// TIA Portal V16 program export: 0 tag tables, 5 data types, 28 data blocks, 30 code blocks (in call order from the OBs), 2 instance data blocks

TYPE "APP"
// stored: IsFailsafeCompliant false
   STRUCT
      PID_ComponenteProporzionale : DInt;
      PID_ComponenteIntegrale : DInt;
      PID_ComponenteDerivativa : DInt;
      Tiro : Int;   // Valore di tiro richiesto: 1-100 => 1-100% Setup 1, 101-200 => 1-100% Setup 2, 0 => Azzera regolatore
      Tiro1 : Int;
      Tiro2 : Int;
      TiroPrecedente : Int;   // Valore di tiro richiesto istante (n-1)
      TiroAppoggio : Int;
      ErroreAttuale : Int;   // Errore istante (n)
      ErrorePrecedente : Int;   // Errore istante (n-1)
      PID_Kp : Int;   // Kp in uso nel PID
      PID_Ki : Int;   // Ki in uso nel PID
      PID_Kd : Int;   // Kd in uso nel PID
      SetpointTiro : Int;   // Valore di setpoint del PID
      SetpointTiroRampa : Int;   // Valore di setpoint del PID iniziale a rampa
      TransitorioInizialeFase1 : Int;   // Indica che si deve eseguire la rampa iniziale (Fase 1)
      TransitorioFase3 : Int;   // Indica che si deve eseguire la rampa da velocita' alta a media (Fase 3)
      TransitorioFase4 : Int;   // Indica che si deve eseguire la rampa da velocita' media a bassa (Fase 4)
      VelocitaRotazione : Int;   // Velocita' di rotazione richiesta
      VelocitaRotazioneFase2 : Int;   // Velocita' di rotazione richiesta durante la Fase 2
      VelocitaRotazioneAppoggio1 : Int;
      VelocitaRotazioneAppoggio2 : Int;
      Fase1OneShoot : Int;   // Indica che sono appena entrato nella fase di traansitorio di accelerazione (Fase 1)
      Fase2OneShoot : Int;   // Indica che sono appena entrato nella fase di transitorio iniziale (Fase 2)
      Fase3OneShoot : Int;   // Indica che sono appena entrato nella fase di transitorio di velocita' alta - media (Fase 3)
      Fase4OneShoot : Int;   // Indica che sono appena entrato nella fase di transitorio di velocita' media - bassa (Fase 4)
      ArrestoRepentinoOneShoot : Int;   // Indica che sono appena entrato nella fase di arresto repentino
      TiroFase1 : Int;   // Indica il tiro nella Fase 1 usato nella Fase 2
      TempIntero : Int;
      Fase : Int;
      BallerinoPrecedente : Array[0..2] of Int;   // Valore del ballerino negli istanti precedenti
      LimiteComponenteIntegrale : Int;   // Limite della componente integrale durante la transizione dalla velocita alta a media (Fase 3) e dalla media a bassa (Fase 4)
      TiroRichiesto : Int;   // Valore di tiro compreso fra 1 e 100 richiesto dalla logica di controllo
      TimerArrestoRepentino : Int;   // Timer per arresto repentino.
      TiroMinimoArrestoRepentino : Int;   // Tiro minimo durante un'arresto repentino
      VariazioneTiro : Int;   // Variazione del tiro film (ballerino)
      TimerFase2 : Int;   // Timer usato nella Fase 2 per arrestare i rulli in caso di rottura film
      TempoRotturaFilm : Int;   // Tempo rottura film in numero di scansioni (1 scansione ogni 30msec)
      TimerFase4 : Int;   // Timer per Fase 4
      TiroMinimoFase4 : Int;   // Tiro minimo durante la Fase 4 di arresto
      PID_Uscita : DInt;   // Valore di uscita del PID
      PrestiroRichiesto : DInt;   // Valore di prestiro richiesto. Valore compreso fra 0 e 500
      PrestiroAppoggio : Real;
   END_STRUCT;
END_TYPE

TYPE "DatiProgramma"
// stored: IsFailsafeCompliant false
   STRUCT
      Wrapping : Bool;   // Wrapping (0=Excluded 1=Included)
      TopLenght : Int;   // Top film lenght
      TopRelease : Int;   // Top carriage release position
      TopDown : Int;   // Top carriage downward to release top film
      Top : Int;   // Top cycle (1=Excluded 2=Before 3=Waterp-2 4=Waterp-3 5=Waterp-4)
      PressurePTime : Int;   // Time for pressure plate downward
      LifterTime : Int;   // Time for pallet lifter upward
      RevOverContrast : Int;   // Revolution over welder contrast
      RopeEndCycle : Byte;   // Rope type at end of cycle (Program)
      Spare4 : Byte;
      RopeTime : Int;   // Delay for rope unit opened
      RevOverClamp : Int;   // Revolution over clamp
      FilmForceFinalRev : Int;   // Film force on the final revolutions
      FilmPrestretchFinalRev : Int;   // Film prestretch on the final revolutions
      ArmSpeed : Int;   // Arm rotation speed (%*10)
      CarriageDown4Top : Int;   // Spool carriage downward for top cycle
      TopDownTime : Int;   // Top carriage downward for top cycle
      LapsUnderTop : Int;   // Revolutions under top film
      Spare6 : Int;   // Spare
      Spare7 : Int;   // Spare
      Spare8 : Int;   // Spare
      Spare9 : Int;   // Spare
      Spare10 : Int;   // Spare
      Spare11 : Int;   // Spare
      Spare12 : Int;   // Spare
      Overlap0_1 : Int := 0;   // Film overlap spool carriage height 0->1
      Height1 : Int := 0;   // Spool carriage height 1 (mm)
      Landmark1 : Bool := false;   // Landmark for spool carriage height 1 (0=Bottom 1=Top)
      Lifter1 : Bool := false;   // Pallet lifter for spool carriage height 1
      SpareBit1H1 : Bool := false;   // Spare bit for spool carriage height 1 (Program)
      Airblower1 : Bool := false;   // Airblower on film tail for spool carriage height 1 (0=Excluded 1=Included)
      NextStep1 : Bool := false;   // Next step for spool carriage height 1 (0=End 1=Next)
      PressureP1 : Bool := false;   // Pressure plate for spool carriage height 1 (0=Excluded 1=Included)
      SpareByte2H1 : Byte := 16#0;   // Spare byte for spool carriage height 1
      Revolution1 : Int := 0;   // Revolutions for spool carriage height 1
      RopeUnit1_1 : Byte := 16#0;   // Rope unit for spool carriage height 1 (1=Excluded 2=Inc 3=Inc during)
      RopeUnit1_2 : Byte := 16#0;   // Rope unit for spool carriage height 1 (1=Excluded 2=Inc 3=Inc during)
      FilmForce1 : Int := 0;   // Film force for spool carriage height 1
      FilmPrestretch1 : Int := 0;   // Film prestretch for spool carriage height 1
      Spare3H1 : Int := 0;   // Spare for spool carriage height 1
      Spare49 : Int := 0;   // Spare
      Spare50 : Int := 0;   // Spare
      Spare51 : Int := 0;   // Spare
      Spare52 : Int := 0;   // Spare
      Spare53 : Int := 0;   // Spare
      Overlap1_2 : Int := 0;   // Film overlap spool carriage height 1->2
      Height2 : Int := 0;   // Spool carriage height 2 (mm)
      Landmark2 : Bool := false;   // Landmark for spool carriage height 2 (0=Bottom 1=Top)
      Lifter2 : Bool := false;   // Pallet lifter for spool carriage height 2
      SpareBit1H2 : Bool := false;   // Spare bit for spool carriage height 2
      Airblower2 : Bool := false;   // Airblower on film tail for spool carriage height 2 (0=Excluded 1=Included)
      NextStep2 : Bool := false;   // Next step for spool carriage height 2 (0=End 1=Next)
      PressureP2 : Bool := false;   // Pressure plate for spool carriage height 2 (0=Excluded 1=Included)
      SpareByte2H2 : Byte := 16#0;   // Spare byte for spool carriage height 2
      Revolution2 : Int := 0;   // Revolutions for spool carriage height 2
      RopeUnit2_1 : Byte := 16#0;   // Rope unit for spool carriage height 2 (1=Excluded 2=Inc 3=Inc during)
      RopeUnit2_2 : Byte := 16#0;   // Rope unit for spool carriage height 2 (1=Excluded 2=Inc 3=Inc during)
      FilmForce2 : Int := 0;   // Film force for spool carriage height 2
      FilmPrestretch2 : Int := 0;   // Film prestretch for spool carriage height 2
      Spare3H2 : Int := 0;   // Spare for spool carriage height 2
      Spare54 : Int := 0;   // Spare
      Spare55 : Int := 0;   // Spare
      Spare56 : Int := 0;   // Spare
      Spare57 : Int := 0;   // Spare
      Spare58 : Int := 0;   // Spare
      Overlap2_3 : Int := 0;   // Film overlap spool carriage height 2->3
      Height3 : Int := 0;   // Spool carriage height 3 (mm)
      Landmark3 : Bool := false;   // Landmark for spool carriage height 3 (0=Bottom 1=Top)
      Lifter3 : Bool := false;   // Pallet lifter for spool carriage height 3
      SpareBit1H3 : Bool := false;   // Spare bit for spool carriage height 3
      Airblower3 : Bool := false;   // Airblower on film tail for spool carriage height 3 (0=Excluded 1=Included)
      NextStep3 : Bool := false;   // Next step for spool carriage height 3 (0=End 1=Next)
      PressureP3 : Bool := false;   // Pressure plate for spool carriage height 3 (0=Excluded 1=Included)
      SpareByte2H3 : Byte := 16#0;   // Spare byte for spool carriage height 3
      Revolution3 : Int := 0;   // Revolutions for spool carriage height 3
      RopeUnit3_1 : Byte := 16#0;   // Rope unit for spool carriage height 3 (1=Excluded 2=Inc 3=Inc during)
      RopeUnit3_2 : Byte := 16#0;   // Rope unit for spool carriage height 3 (1=Excluded 2=Inc 3=Inc during)
      FilmForce3 : Int := 0;   // Film force for spool carriage height 3
      FilmPrestretch3 : Int := 0;   // Film prestretch for spool carriage height 3
      Spare3H3 : Int := 0;   // Spare for spool carriage height 3
      Spare59 : Int := 0;   // Spare
      Spare60 : Int := 0;   // Spare
      Spare61 : Int := 0;   // Spare
      Spare62 : Int := 0;   // Spare
      Spare63 : Int := 0;   // Spare
      Overlap3_4 : Int := 0;   // Film overlap spool carriage height 3->4
      Height4 : Int := 0;   // Spool carriage height 4 (mm)
      Landmark4 : Bool := false;   // Landmark for spool carriage height 4 (0=Bottom 1=Top)
      Lifter4 : Bool := false;   // Pallet lifter for spool carriage height 4
      SpareBit1H4 : Bool := false;   // Spare bit for spool carriage height 4
      Airblower4 : Bool := false;   // Airblower on film tail for spool carriage height 4 (0=Excluded 1=Included)
      NextStep4 : Bool := false;   // Next step for spool carriage height 4 (0=End 1=Next)
      PressureP4 : Bool := false;   // Pressure plate for spool carriage height 4 (0=Excluded 1=Included)
      SpareByte2H4 : Byte := 16#0;   // Spare byte for spool carriage height 4
      Revolution4 : Int := 0;   // Revolutions for spool carriage height 4
      RopeUnit4_1 : Byte := 16#0;   // Rope unit for spool carriage height 4 (1=Excluded 2=Inc 3=Inc during)
      RopeUnit4_2 : Byte := 16#0;   // Rope unit for spool carriage height 4 (1=Excluded 2=Inc 3=Inc during)
      FilmForce4 : Int := 0;   // Film force for spool carriage height 4
      FilmPrestretch4 : Int := 0;   // Film prestretch for spool carriage height 4
      Spare3H4 : Int := 0;   // Spare for spool carriage height 4
      Spare64 : Int := 0;   // Spare
      Spare65 : Int := 0;   // Spare
      Spare66 : Int := 0;   // Spare
      Spare67 : Int := 0;   // Spare
      Spare68 : Int := 0;   // Spare
      Overlap4_5 : Int := 0;   // Film overlap spool carriage height 4->5
      Height5 : Int := 0;   // Spool carriage height 5 (mm)
      Landmark5 : Bool := false;   // Landmark for spool carriage height 5 (0=Bottom 1=Top)
      Lifter5 : Bool := false;   // Pallet lifter for spool carriage height 5
      SpareBit1H5 : Bool := false;   // Spare bit for spool carriage height 5
      Airblower5 : Bool := false;   // Airblower on film tail for spool carriage height 5 (0=Excluded 1=Included)
      NextStep5 : Bool := false;   // Next step for spool carriage height 5 (0=End 1=Next)
      PressureP5 : Bool := false;   // Pressure plate for spool carriage height 5 (0=Excluded 1=Included)
      SpareByte2H5 : Byte := 16#0;   // Spare byte for spool carriage height 5
      Revolution5 : Int := 0;   // Revolutions for spool carriage height 5
      RopeUnit5_1 : Byte := 16#0;   // Rope unit for spool carriage height 5 (1=Excluded 2=Inc 3=Inc during)
      RopeUnit5_2 : Byte := 16#0;   // Rope unit for spool carriage height 5 (1=Excluded 2=Inc 3=Inc during)
      FilmForce5 : Int := 0;   // Film force for spool carriage height 5
      FilmPrestretch5 : Int := 0;   // Film prestretch for spool carriage height 5
      Spare3H5 : Int := 0;   // Spare for spool carriage height 5
      Spare69 : Int := 0;   // Spare
      Spare70 : Int := 0;   // Spare
      Spare71 : Int := 0;   // Spare
      Spare72 : Int := 0;   // Spare
      Spare73 : Int := 0;   // Spare
      Overlap5_6 : Int := 0;   // Film overlap spool carriage height 5->6
      Height6 : Int := 0;   // Spool carriage height 6 (mm)
      Landmark6 : Bool := false;   // Landmark for spool carriage height 6 (0=Bottom 1=Top)
      Lifter6 : Bool := false;   // Pallet lifter for spool carriage height 6
      SpareBit1H6 : Bool := false;   // Spare bit for spool carriage height 6
      Airblower6 : Bool := false;   // Airblower on film tail for spool carriage height 6 (0=Excluded 1=Included)
      NextStep6 : Bool := false;   // Next step for spool carriage height 6 (0=End 1=Next)
      PressureP6 : Bool := false;   // Pressure plate for spool carriage height 6 (0=Excluded 1=Included)
      SpareByte2H6 : Byte := 16#0;   // Spare byte for spool carriage height 6
      Revolution6 : Int := 0;   // Revolutions for spool carriage height 6
      RopeUnit6_1 : Byte := 16#0;   // Rope unit for spool carriage height 6 (1=Excluded 2=Inc 3=Inc during)
      RopeUnit6_2 : Byte := 16#0;   // Rope unit for spool carriage height 6 (1=Excluded 2=Inc 3=Inc during)
      FilmForce6 : Int := 0;   // Film force for spool carriage height 6
      FilmPrestretch6 : Int := 0;   // Film prestretch for spool carriage height 6
      Spare3H6 : Int := 0;   // Spare for spool carriage height 6
      Spare74 : Int := 0;   // Spare
      Spare75 : Int := 0;   // Spare
      Spare76 : Int := 0;   // Spare
      Spare77 : Int := 0;   // Spare
      Spare78 : Int := 0;   // Spare
      Overlap6_7 : Int := 0;   // Film overlap spool carriage height 6->7
      Height7 : Int := 0;   // Spool carriage height 7 (mm)
      Landmark7 : Bool := false;   // Landmark for spool carriage height 7 (0=Bottom 1=Top)
      Lifter7 : Bool := false;   // Pallet lifter for spool carriage height 7
      SpareBit1H7 : Bool := false;   // Spare bit for spool carriage height 7
      Airblower7 : Bool := false;   // Airblower on film tail for spool carriage height 7 (0=Excluded 1=Included)
      NextStep7 : Bool := false;   // Next step for spool carriage height 7 (0=End 1=Next)
      PressureP7 : Bool := false;   // Pressure plate for spool carriage height 7 (0=Excluded 1=Included)
      SpareByte2H7 : Byte := 16#0;   // Spare byte for spool carriage height 7
      Revolution7 : Int := 0;   // Revolutions for spool carriage height 7
      RopeUnit7_1 : Byte := 16#0;   // Rope unit for spool carriage height 7 (1=Excluded 2=Inc 3=Inc during)
      RopeUnit7_2 : Byte := 16#0;   // Rope unit for spool carriage height 7 (1=Excluded 2=Inc 3=Inc during)
      FilmForce7 : Int := 0;   // Film force for spool carriage height 7
      FilmPrestretch7 : Int := 0;   // Film prestretch for spool carriage height 7
      Spare3H7 : Int := 0;   // Spare for spool carriage height 7
      Spare79 : Int := 0;   // Spare
      Spare80 : Int := 0;   // Spare
      Spare81 : Int := 0;   // Spare
      Spare82 : Int := 0;   // Spare
      Spare83 : Int := 0;   // Spare
      Overlap7_8 : Int := 0;   // Film overlap spool carriage height 7->8
      Height8 : Int := 0;   // Spool carriage height 8 (mm)
      Landmark8 : Bool := false;   // Landmark for spool carriage height 8 (0=Bottom 1=Top)
      Lifter8 : Bool := false;   // Pallet lifter for spool carriage height 8
      SpareBit1H8 : Bool := false;   // Spare bit for spool carriage height 8
      Airblower8 : Bool := false;   // Airblower on film tail for spool carriage height 8 (0=Excluded 1=Included)
      NextStep8 : Bool := false;   // Next step for spool carriage height 8 (0=End 1=Next)
      PressureP8 : Bool := false;   // Pressure plate for spool carriage height 8 (0=Excluded 1=Included)
      SpareByte2H8 : Byte := 16#0;   // Spare byte for spool carriage height 8
      Revolution8 : Int := 0;   // Revolutions for spool carriage height 8
      RopeUnit8_1 : Byte := 16#0;   // Rope unit for spool carriage height 8 (1=Excluded 2=Inc 3=Inc during)
      RopeUnit8_2 : Byte := 16#0;   // Rope unit for spool carriage height 8 (1=Excluded 2=Inc 3=Inc during)
      FilmForce8 : Int := 0;   // Film force for spool carriage height 8
      FilmPrestretch8 : Int := 0;   // Film prestretch for spool carriage height 8
      Spare3H8 : Int := 0;   // Spare for spool carriage height 8
      Spare84 : Int := 0;   // Spare
      Spare85 : Int := 0;   // Spare
      Spare86 : Int := 0;   // Spare
      Spare87 : Int := 0;   // Spare
      Spare88 : Int := 0;   // Spare
      Overlap8_9 : Int := 0;   // Film overlap spool carriage height 8->9
      Height9 : Int := 0;   // Spool carriage height 9 (mm)
      Landmark9 : Bool := false;   // Landmark for spool carriage height 9 (0=Bottom 1=Top)
      Lifter9 : Bool := false;   // Pallet lifter for spool carriage height 9
      SpareBit1H9 : Bool := false;   // Spare bit for spool carriage height 9
      Airblower9 : Bool := false;   // Airblower on film tail for spool carriage height 9 (0=Excluded 1=Included)
      NextStep9 : Bool := false;   // Next step for spool carriage height 9 (0=End 1=Next)
      PressureP9 : Bool := false;   // Pressure plate for spool carriage height 9 (0=Excluded 1=Included)
      SpareByte2H9 : Byte := 16#0;   // Spare byte for spool carriage height 9
      Revolution9 : Int := 0;   // Revolutions for spool carriage height 9
      RopeUnit9_1 : Byte := 16#0;   // Rope unit for spool carriage height 9 (1=Excluded 2=Inc 3=Inc during)
      RopeUnit9_2 : Byte := 16#0;   // Rope unit for spool carriage height 9 (1=Excluded 2=Inc 3=Inc during)
      FilmForce9 : Int := 0;   // Film force for spool carriage height 9
      FilmPrestretch9 : Int := 0;   // Film prestretch for spool carriage height 9
      Spare3H9 : Int := 0;   // Spare for spool carriage height 9
      Spare89 : Int := 0;   // Spare
      Spare90 : Int := 0;   // Spare
      Spare91 : Int := 0;   // Spare
      Spare92 : Int := 0;   // Spare
      Spare93 : Int := 0;   // Spare
      Overlap9_10 : Int := 0;   // Film overlap spool carriage height 9->10
      Height10 : Int := 0;   // Spool carriage height 10 (mm)
      Landmark10 : Bool := false;   // Landmark for spool carriage height 10 (0=Bottom 1=Top)
      Lifter10 : Bool := false;   // Pallet lifter for spool carriage height 10
      SpareBit1H10 : Bool := false;   // Spare bit for spool carriage height 10
      Airblower10 : Bool := false;   // Airblower on film tail for spool carriage height 10 (0=Excluded 1=Included)
      NextStep10 : Bool := false;   // Next step for spool carriage height 10 (0=End 1=Next)
      PressureP10 : Bool := false;   // Pressure plate for spool carriage height 10 (0=Excluded 1=Included)
      SpareByte2H10 : Byte := 16#0;   // Spare byte for spool carriage height 10
      Revolution10 : Int := 0;   // Revolutions for spool carriage height 10
      RopeUnit10_1 : Byte := 16#0;   // Rope unit for spool carriage height 10 (1=Excluded 2=Inc 3=Inc during)
      RopeUnit10_2 : Byte := 16#0;   // Rope unit for spool carriage height 10 (1=Excluded 2=Inc 3=Inc during)
      FilmForce10 : Int := 0;   // Film force for spool carriage height 10
      FilmPrestretch10 : Int := 0;   // Film prestretch for spool carriage height 10
      Spare3H10 : Int := 0;   // Spare for spool carriage height 10
      Spare94 : Int := 0;   // Spare
      Spare95 : Int := 0;   // Spare
      Spare96 : Int := 0;   // Spare
      Spare97 : Int := 0;   // Spare
      Spare98 : Int := 0;   // Spare
      Overlap10_11 : Int := 0;   // Film overlap spool carriage height 10->11
      Height11 : Int := 0;   // Spool carriage height 11 (mm)
      Landmark11 : Bool := false;   // Landmark for spool carriage height 11 (0=Bottom 1=Top)
      Lifter11 : Bool := false;   // Pallet lifter for spool carriage height 11
      SpareBit1H11 : Bool := false;   // Spare bit for spool carriage height 11
      Airblower11 : Bool := false;   // Airblower on film tail for spool carriage height 11 (0=Excluded 1=Included)
      NextStep11 : Bool := false;   // Next step for spool carriage height 11 (0=End 1=Next)
      PressureP11 : Bool := false;   // Pressure plate for spool carriage height 11 (0=Excluded 1=Included)
      SpareByte2H11 : Byte := 16#0;   // Spare byte for spool carriage height 11
      Revolution11 : Int := 0;   // Revolutions for spool carriage height 11
      RopeUnit11_1 : Byte := 16#0;   // Rope unit for spool carriage height 11 (1=Excluded 2=Inc 3=Inc during)
      RopeUnit11_2 : Byte := 16#0;   // Rope unit for spool carriage height 11 (1=Excluded 2=Inc 3=Inc during)
      FilmForce11 : Int := 0;   // Film force for spool carriage height 11
      FilmPrestretch11 : Int := 0;   // Film prestretch for spool carriage height 11
      Spare3H11 : Int := 0;   // Spare for spool carriage height 11
      Spare99 : Int := 0;   // Spare
      Spare100 : Int := 0;   // Spare
      Spare101 : Int := 0;   // Spare
      Spare102 : Int := 0;   // Spare
      Spare103 : Int := 0;   // Spare
      Overlap11_12 : Int := 0;   // Film overlap spool carriage height 11->12
      Height12 : Int := 0;   // Spool carriage height 12 (mm)
      Landmark12 : Bool := false;   // Landmark for spool carriage height 12 (0=Bottom 1=Top)
      Lifter12 : Bool := false;   // Pallet lifter for spool carriage height 12
      SpareBit1H12 : Bool := false;   // Spare bit for spool carriage height 12
      Airblower12 : Bool := false;   // Airblower on film tail for spool carriage height 12 (0=Excluded 1=Included)
      NextStep12 : Bool := false;   // Next step for spool carriage height 12 (0=End 1=Next)
      PressureP12 : Bool := false;   // Pressure plate for spool carriage height 12 (0=Excluded 1=Included)
      SpareByte2H12 : Byte := 16#0;   // Spare byte for spool carriage height 12
      Revolution12 : Int := 0;   // Revolutions for spool carriage height 12
      RopeUnit12_1 : Byte := 16#0;   // Rope unit for spool carriage height 12 (1=Excluded 2=Inc 3=Inc during)
      RopeUnit12_2 : Byte := 16#0;   // Rope unit for spool carriage height 12 (1=Excluded 2=Inc 3=Inc during)
      FilmForce12 : Int := 0;   // Film force for spool carriage height 12
      FilmPrestretch12 : Int := 0;   // Film prestretch for spool carriage height 12
      Spare3H12 : Int := 0;   // Spare for spool carriage height 12
      Spare104 : Int := 0;   // Spare
      Spare105 : Int := 0;   // Spare
      Spare106 : Int := 0;   // Spare
      Spare107 : Int := 0;   // Spare
      Spare108 : Int := 0;   // Spare
   END_STRUCT;
END_TYPE

TYPE "M20"
// stored: IsFailsafeCompliant false
   STRUCT
      M20_P00 : Int;   // Tipo di prestiro
      M20_P01 : Int;   // Coefficiente proporzionale per il regolatore PID
      M20_P02 : Int;   // Coefficiente integrale (Fase1 e Fase2) per il regolatore PID
      M20_P03 : Int;   // Coefficiente derivativo per il regolatore PID
      M20_P04 : Int;   // Coefficiente integrale (Fase3 e Fase4) per il regolatore PID
      M20_P05 : Int;   // Rampa di accelerazione per il tiro durante la Fase1
      M20_P06 : Int;   // Limite componente integrale nel transitorio dalla Fase2 alla Fase3
      M20_P07 : Int;   // Limite componente integrale nel transitorio dalla Fase3 alla Fase4
      M20_P08 : Int;   // Valore minimo ingresso analogico
      M20_P09 : Int;   // Valore massimo ingresso analogico
      M20_P10 : Int;   // Prestiro naturale dovuto al rapporto di riduzione
      M20_P11 : Int;   // Velocità per il jog in manuale dei rulli di prestiro
      M20_P12 : Int;   // Offset del rullo lento 10 equivale a 0
      M20_P13 : Int;   // Jog di velocità durante la partenza del braccio
      M20_P14 : Int;   // Tiro minimo durante la Fase4 di arresto e durante un arresto repentino
      M20_P15 : Int;   // Tempo (in decimi di secondo) dopo il quale i rulli si fermano per rottura film
      M20_P20 : Int;   // Velocità indicata da plc per la rotazione braccio e il carrello top
      M20_P21 : Int;   // Velocità indicata da plc per il carrello di prestiro e il trasporto di centro macchina
      M20_P22 : Int;   // Tiro indicato da plc
      M20_P23 : Int;   // Prestiro indicato da plc
      M20_P24 : Int;   // Valore di ingresso analogico AI0
      M20_P25 : Int;   // Tiro richiesto da plc compreso fra 0 e 100
   END_STRUCT;
END_TYPE

TYPE "PID"
// stored: IsFailsafeCompliant false
   STRUCT
      proporzionale : DInt;
      integrativo : DInt;
      segnale : DInt;
      maxSegnale : Int;
      minSegnale : Int;
      setPointShow : UInt;
      tiro : UInt;
      vParP : UInt;
      vParI : UInt;
      svuota : Bool;
      attiva : Bool;
      setTiro : Bool;
      "timer" : Time;
   END_STRUCT;
END_TYPE

TYPE "ProgramDataGreyBar"
// stored: IsFailsafeCompliant false
   STRUCT
      Overlap : Int;   // Film overlap
      Height : Int;   // Spool carriage height (mm)
      Landmark : Bool;   // Landmark (0=Bottom 1=Top)
      Lifter : Bool;   // Pallet lifter
      SpareBit1 : Bool;   // Spare
      Airblower : Bool;   // Airblower on film tail (0=Excluded 1=Included)
      NextStep : Bool;   // Next step (0=End 1=Next)
      PressureP : Bool;   // Pressure plate (0=Excluded 1=Included)
      SpareByte1 : Byte;   // Spare
      Revolution : Int;   // Revolutions
      RopeUnitUpper : Byte;   // Upper rope unit (1=Exc 2=Inc 3=Inc during)
      RopeUnitLower : Byte;   // Lower rope unit (1=Exc 2=Inc 3=Inc during)
      FilmForce : Int;   // Film force
      FilmPrestretch : Int;   // Film prestretch
      SpareWord1 : Int;   // Spare
      SpareWord2 : Int;   // Spare
      SpareWord3 : Int;   // Spare
      SpareWord4 : Int;   // Spare
      SpareWord5 : Int;   // Spare
      SpareWord6 : Int;   // Spare
   END_STRUCT;
END_TYPE

DATA_BLOCK "DB01_Osr"   // DB1
{ S7_Optimized_Access := 'FALSE' }
AUTHOR : Robopac
VERSION : 0.0
// stored: AutoNumber false, IsOnlyStoredInLoadMemory false, IsWriteProtectedInAS false
   VAR RETAIN
      osr1 : Bool := TRUE;   // Used
      osr2 : Bool := FALSE;   // Used
      osr3 : Bool := FALSE;   // Used
      osr4 : Bool := FALSE;   // Used
      osr5 : Bool := FALSE;   // Used
      osr6 : Bool := TRUE;   // Used
      osr7 : Bool := TRUE;   // Used
      osr8 : Bool := FALSE;   // Used
      osr9 : Bool := TRUE;   // Used
      osr10 : Bool := FALSE;   // Used
      osr11 : Bool := FALSE;   // Used
      osr12 : Bool := FALSE;   // Used
      osr13 : Bool := FALSE;   // Used
      osr14 : Bool := FALSE;   // Used
      osr15 : Bool := TRUE;   // Used
      osr16 : Bool := FALSE;   // Used
      osr17 : Bool := TRUE;   // Used
      osr18 : Bool := TRUE;   // Used
      osr19 : Bool := TRUE;   // Used
      osr20 : Bool := TRUE;   // Used
      osr21 : Bool := TRUE;   // Used
      osr22 : Bool := TRUE;   // Used
      osr23 : Bool := FALSE;   // Used
      osr24 : Bool := FALSE;   // Used
      osr25 : Bool := FALSE;   // Used
      osr26 : Bool := FALSE;   // Used
      osr27 : Bool := FALSE;   // Used
      osr28 : Bool := FALSE;   // Used
      osr29 : Bool := FALSE;   // Used
      osr30 : Bool := TRUE;   // Used
      osr31 : Bool := TRUE;   // Used
      osr32 : Bool := TRUE;   // Used
      osr33 : Bool := TRUE;   // Used
      osr34 : Bool := TRUE;   // Used
      osr35 : Bool := FALSE;   // Used
      osr36 : Bool := FALSE;   // Used
      osr37 : Bool := TRUE;
      osr38 : Bool := FALSE;   // Used
      osr39 : Bool := TRUE;   // Used
      osr40 : Bool := FALSE;   // Used
      osr41 : Bool := TRUE;   // Used
      osr42 : Bool := TRUE;
      osr43 : Bool := TRUE;
      osr44 : Bool := FALSE;
      osr45 : Bool := FALSE;   // Used
      osr46 : Bool := FALSE;   // Used
      osr47 : Bool := FALSE;
      osr48 : Bool := FALSE;
      osr49 : Bool := FALSE;
      osr50 : Bool := TRUE;
      osr51 : Bool := FALSE;
      osr52 : Bool := TRUE;
      osr53 : Bool := FALSE;
      osr54 : Bool := FALSE;
      osr55 : Bool := FALSE;
      osr56 : Bool := TRUE;
      osr57 : Bool := FALSE;
      osr58 : Bool := FALSE;
      osr59 : Bool := FALSE;
      osr60 : Bool := TRUE;
      osr61 : Bool := FALSE;
      osr62 : Bool := FALSE;
      osr63 : Bool := FALSE;
      osr64 : Bool := FALSE;
      osr65 : Bool := FALSE;
      osr66 : Bool := FALSE;
      osr67 : Bool := TRUE;
      osr68 : Bool := FALSE;
      osr69 : Bool := TRUE;
      osr70 : Bool := FALSE;
      osr71 : Bool := FALSE;
      osr72 : Bool := FALSE;
      osr73 : Bool := FALSE;
      osr74 : Bool := TRUE;
      osr75 : Bool := TRUE;
      osr76 : Bool := FALSE;
      osr77 : Bool := TRUE;
      osr78 : Bool := TRUE;
      osr79 : Bool := FALSE;
      osr80 : Bool := FALSE;
      osr81 : Bool := FALSE;   // Used
      osr82 : Bool := FALSE;   // Used
      osr83 : Bool := FALSE;
      osr84 : Bool := FALSE;
      osr85 : Bool := FALSE;
      osr86 : Bool := FALSE;
      osr87 : Bool := FALSE;
      osr88 : Bool := TRUE;
      osr89 : Bool := FALSE;
      osr90 : Bool := FALSE;   // Used
      osr91 : Bool := FALSE;
      osr92 : Bool := FALSE;
      osr93 : Bool := TRUE;
      osr94 : Bool := TRUE;
      osr95 : Bool := TRUE;
      osr96 : Bool := TRUE;
   END_VAR
BEGIN
END_DATA_BLOCK

DATA_BLOCK "DB03_Machine"   // DB3
{ S7_Optimized_Access := 'FALSE' }
AUTHOR : Robopac
VERSION : 0.0
// stored: AutoNumber false, IsOnlyStoredInLoadMemory false, IsWriteProtectedInAS false
   VAR RETAIN
      dbx0_0 : Bool := FALSE;   // Enable the arm rotation revolution counter
      dbx0_1 : Bool := FALSE;   // High pressure on prestretch roller dancer
      dbx0_2 : Bool := FALSE;   // One arm revolution done support memory
      dbx0_3 : Bool := FALSE;   // One arm revolution done
      dbx0_4 : Bool := FALSE;   // Support memory for revolution counter
      dbx0_5 : Bool := FALSE;   // Support memory for 10% prestretch carriage
      dbx0_6 : Bool := FALSE;
      dbx0_7 : Bool := FALSE;   // Support memory for arm rotation speed recorded
      dbb1 : Byte := 16#00;
      MachineExc : Bool := FALSE;   // Wrapping excluded
      MachineInc : Bool := FALSE;   // Wrapping included
      dbb3 : Byte := 16#00;
      dbx4_0 : Bool := FALSE;   // Memory to silent acoustic signal on alarm
      dbx4_1 : Bool := FALSE;
      dbx4_2 : Bool := FALSE;   // Condition to check all out of positon alarm
      dbx4_3 : Bool := FALSE;   // Condition for manual operation
      dbx4_4 : Bool := FALSE;   // All units are ready for automatic cycle
      dbx4_5 : Bool := FALSE;
      dbx4_6 : Bool := FALSE;   // Data for next ring height loaded
      dbx4_7 : Bool := FALSE;   // Data for next ring height loaded
      dbx5_0 : Bool := FALSE;   // Wrapping cycle: Next step is cut and pallet unload
      dbx5_1 : Bool := FALSE;   // Wrapping cycle: Next step is cut and new spool carriage height
      dbx5_2 : Bool := FALSE;   // Wrapping cycle: Next step is new spool carriage height
      dbx5_3 : Bool := FALSE;   // Wrapping cycle: After this step top waterproof
      dbx5_4 : Bool := FALSE;   // Wrong data program for the pallet on the machine
      dbx5_5 : Bool := FALSE;   // Closing upper(double) rope unit
      dbx5_6 : Bool := FALSE;   // Closing single or lower(double) rope unit
      dbx5_7 : Bool := FALSE;   // Memory for timeout enable
      dbx6_0 : Bool := FALSE;   // Memory to exclude infeed safety barrier
      dbx6_1 : Bool := FALSE;   // Memory to exclude outfeed safety barrier
      dbx6_2 : Bool := FALSE;   // Memory to exclude infeed safety barrier
      dbx6_3 : Bool := FALSE;   // Memory to exclude infeed safety barrier
      dbx6_4 : Bool := FALSE;   // Memory to exclude outfeed safety barrier
      dbx6_5 : Bool := FALSE;   // Memory to exclude outfeed safety barrier
      dbx6_6 : Bool := FALSE;
      dbx6_7 : Bool := FALSE;
      dbx7_0 : Bool := FALSE;   // Pressure plate excluded for low pallet
      dbx7_1 : Bool := FALSE;
      dbx7_2 : Bool := FALSE;   // Support memory to check rotation speed
      dbx7_3 : Bool := FALSE;   // Support memory to check spool carriage speed
      dbx7_4 : Bool := FALSE;   // Used by S7-200
      dbx7_5 : Bool := FALSE;   // Machine in wrapping cycle
      dbx7_6 : Bool := FALSE;   // Support memory to refresh pallet per hour value
      dbx7_7 : Bool := FALSE;
      dbb8 : Byte := 16#00;
      TopExc : Bool := FALSE;   // Top excluded
      TopBefore : Bool := FALSE;   // Top included before wrapping beginning
      TopWaterP : Bool := FALSE;   // Top included waterproof
      dbw10 : Int := 0;
      dbw12 : Int := 0;   // Counter for revolution on running spool carriage height
      dbw14 : Int := 0;   // Counter for revolution on welder contrast
      dbw16 : Int := 0;   // Counter for revolution of deceleration
      dbw18 : Int := 0;
      dbw20 : Int := 0;   // Active program for multiprogram (Display)
      dbw22 : Int := 0;   // Selected program for multiprogram (Display)
      dbw24 : Int := 0;   // Program to be shown on data program page (Display)
      dbw26 : Int := 0;   // Program selection by external signal
      dbw28 : Int := 0;   // Program selection by external signal
      dbw30 : Int := 0;   // Support memory for data transfer
      dbw32 : Int := 0;   // Arm rotation speed recorded (rpm*10)
      dbw34 : Int := 0;   // Required arm rotation speed recorded (%*10)
      dbw36 : Int := 0;
      dbw38 : Int := 0;   // Support memory to evaluate carriage movement speed
      dbw40 : Int := 0;   // Support memory to evaluate carriage movement speed
      dbw42 : Int := 0;   // Spool carriage movement speed mm/sec
      dbw44 : Int := 0;   // table rotation movement speed mm/sec
      dbw46 : Int := 0;   // Arm rotation speed (rpm*10) related to actual required speed
      dbw48 : Int := 0;   // Spool carriage movement speed mm/sec recorded
      dbw50 : Int := 0;
      dbw52 : Int := 0;   // High speed for spool carriage movement (%) recorded from display
      dbw54 : Int := 0;   // upport memory for spool carriage high speed
      dbw56 : Int := 0;   // Spool carriage movement speed used on cycle (mm/sec)
      dbb58 : Byte := 16#00;   // Counter for DAC M20 converter
      dbx59_0 : Bool := FALSE;   // Arm rotation and top carriage speed change for DAC M20
      dbx59_1 : Bool := FALSE;   // Spool carriage speed change for DAC M20
      dbx59_2 : Bool := FALSE;   // Counter for DAC M20 is odd
      dbx59_3 : Bool := FALSE;
      dbx59_4 : Bool := FALSE;
      dbx59_5 : Bool := FALSE;
      dbx59_6 : Bool := FALSE;
      dbx59_7 : Bool := FALSE;
      dbw60 : Int := 0;   // Value for DAC analog output
      dbw62 : Int := 0;
      dbw64 : Int := 0;
      dbw66 : Int := 0;   // Support for running height data transfer
      dbw68 : Int := 0;   // Number of the running spool carriage height
      dbw70 : Int := 0;   // Film overlap for running spool carriage height
      dbw72 : Int := 0;   // Carriage height (mm) for running spool carriage height
      dbx74_0 : Bool := FALSE;   // Landmark (0=Bottom 1=Top) for running spool carriage height
      dbx74_1 : Bool := FALSE;   // Pallet lifter for running spool carriage height (0=Excluded 1=Included)
      dbx74_2 : Bool := FALSE;   // Spare
      dbx74_3 : Bool := FALSE;   // Airblower on film tail for running spool carriage height (0=Exc 1=Inc)
      dbx74_4 : Bool := FALSE;   // Next step for running spool carriage height (0=End 1=Next)
      dbx74_5 : Bool := FALSE;   // Pressure plate for running spool carriage height (0=Excluded 1=Included)
      dbx74_6 : Bool := FALSE;   // Spare
      dbx74_7 : Bool := FALSE;   // Spare
      dbb75 : Byte := 16#00;   // Spare
      dbw76 : Int := 0;   // Revolutions for running spool carriage height
      dbb78 : Byte := 16#00;   // Rope unit for running spool carriage height (1=Excluded 2=Inc 3=Inc during)
      dbb79 : Byte := 16#00;   // Rope unit for running spool carriage height (1=Excluded 2=Inc 3=Inc during)
      dbw80 : Int := 0;   // Film force for running spool carriage height
      dbw82 : Int := 0;   // Film prestretch for running spool carriage height
      dbw84 : Int := 0;   // Delay to open or close upper rope unit for runninh spool carriage height
      dbw86 : Int := 0;   // Delay to open or close lower rope unit for runninh spool carriage height
      dbw88 : Int := 0;   // Spare for running spool carriage height
      dbw90 : Int := 0;   // Spare for running spool carriage height
      dbw92 : Int := 0;   // Spare for running spool carriage height
      dbw94 : Int := 0;   // Spare for running spool carriage height
      dbw96 : Int := 0;
      dbw98 : Int := 0;
   END_VAR
BEGIN
END_DATA_BLOCK

DATA_BLOCK "DB05_SpoolCarriagePos"   // DB5
{ S7_Optimized_Access := 'FALSE' }
AUTHOR : Robopac
VERSION : 0.0
// stored: AutoNumber false, IsOnlyStoredInLoadMemory false, IsWriteProtectedInAS false
   VAR RETAIN
      dbx0_0 : Bool := FALSE;   // Table rotation forward
      dbx0_1 : Bool := FALSE;   // Table rotation backward
      dbx0_2 : Bool := FALSE;   // Table rotation speed: Low
      dbx0_3 : Bool := FALSE;   // Table rotation speed: Middle 1 for top
      dbx0_4 : Bool := FALSE;   // Table rotation speed: Middle 2 for welder contrast
      dbx0_5 : Bool := FALSE;   // Table rotation speed: High
      dbx0_6 : Bool := FALSE;
      dbx0_7 : Bool := FALSE;
      dbx1_0 : Bool := FALSE;   // Spool carriage axis movement upward
      dbx1_1 : Bool := FALSE;   // Spool carriage axis movement downward
      dbx1_2 : Bool := FALSE;   // Spool carriage axis movement inside low speed area
      dbx1_3 : Bool := FALSE;   // Spool carriage axis movement low speed
      dbx1_4 : Bool := FALSE;   // Spool carriage upward
      dbx1_5 : Bool := FALSE;   // Spool carriage downward
      dbx1_6 : Bool := FALSE;
      dbx1_7 : Bool := FALSE;
      dbx2_0 : Bool := FALSE;
      dbx2_1 : Bool := FALSE;   // Support memory for enable (EN) on table rotation and table conveyor inverter
      dbx2_2 : Bool := FALSE;
      dbx2_3 : Bool := FALSE;
      dbx2_4 : Bool := FALSE;
      dbx2_5 : Bool := FALSE;
      dbx2_6 : Bool := FALSE;
      dbx2_7 : Bool := FALSE;
      dbx3_0 : Bool := FALSE;   // Spool carriage: Support for encoder running control
      dbx3_1 : Bool := FALSE;   // Spool carriage: Support for encoder running control alarm
      dbx3_2 : Bool := FALSE;
      dbx3_3 : Bool := FALSE;
      dbx3_4 : Bool := FALSE;
      dbx3_5 : Bool := FALSE;
      dbx3_6 : Bool := FALSE;
      dbx3_7 : Bool := FALSE;
      dbx4_0 : Bool := FALSE;   // Pallet height recording in automatic mode
      dbx4_1 : Bool := FALSE;   // Support memory for pallet height recording
      dbx4_2 : Bool := FALSE;
      dbx4_3 : Bool := FALSE;   // Support memory for pallet height filter
      dbx4_4 : Bool := FALSE;   // Condition for pallet height detected
      dbx4_5 : Bool := FALSE;
      dbx4_6 : Bool := TRUE;   // Carriage in position to rotate in medium to wrap top
      dbx4_7 : Bool := FALSE;
      dbx5_0 : Bool := FALSE;
      dbx5_1 : Bool := FALSE;
      dbx5_2 : Bool := FALSE;
      dbx5_3 : Bool := FALSE;
      dbx5_4 : Bool := TRUE;   // Top wrapped ring position
      dbw6 : Int := 100;   // Spool carriage: Support for movement speed
      dbw8 : Int := 50;   // Spool carriage: Support for movement deceleration
      dbw10 : Int := 100;
      dbw12 : Int := 10199;
      dbw14 : Int := 10306;   // Pallet height on machine conveyor + 300 mm
      dbw16 : Int := 9999;   // Pallet height on machine conveyor
      dbw18 : Int := 9999;   // Pallet height on machine conveyor
      dbw20 : Int := 480;   // Spool carriage height for middle speed on welder contrast
      dbw22 : Int := -2;   // Support memory for pallet height filter
      dbw24 : Int := 0;   // Support memory for pallet height
      dbw26 : Int := -380;   // Spool carriage height for middle speed before top cycle
      dbw28 : Int := 0;
      dbd30 : DInt := -1;   // Spool carriage position: Pulse
      dbw34 : Int := -2;   // Spool carriage position: Top of the spool
      dbw36 : Int := 1782;   // Spool carriage position: Spool carriage all up position
      dbw38 : Int := 50;   // Spool carriage position: Deceleration position for carriage overrun down
      dbw40 : Int := 1732;   // Spool carriage position: Deceleration position for carriage overrun up
      dbd42 : DInt := -1;   // Support for encoder spool carriage running control
      dbw46 : Int := 12;   // Support for encoder spool carriage running control
      dbw48 : Int := 0;
      dbw50 : Int := 0;   // Support memory for machine conveyor speed (%)
      dbw52 : Int := 0;   // Support memory for spool carriage and machine conveyor speed (%)
      dbw54 : Int := 0;   // Support memory for for arm rotation speed (%*10)
      dbw56 : Int := 0;   // Support memory for top carriage forward/backward speed (%*10)
      dbw58 : Int := 0;   // Support memory for top carriage forward/backward and arm rotation speed (%*10)
      dbw60 : Int := 0;
      dbw62 : Int := 0;
      dbw64 : Int := 0;
      dbw66 : Int := 0;
      dbw68 : Int := 0;
      Req1_Start : Bool := FALSE;   // Positioning request 1: Start
      Req2_Start : Bool := FALSE;   // Positioning request 2: Start
      Req3_Start : Bool := FALSE;   // Positioning request 3: Start
      Req4_Start : Bool := FALSE;   // Positioning request 4: Start
      Req5_Start : Bool := FALSE;   // Positioning request 5: Start
      Req6_Start : Bool := FALSE;   // Positioning request 6: Start
      Req7_Start : Bool := FALSE;   // Positioning request 7: Start
      Req8_Start : Bool := FALSE;   // Positioning request 8: Start
      Req9_Start : Bool := FALSE;   // Positioning request 9: Start
      Req10_Start : Bool := FALSE;   // Positioning request 10: Start
      Req1_Dest : Int := 50;   // Positioning request 1: Destination position
      Req2_Dest : Int := 40;   // Positioning request 2: Destination position
      Req3_Dest : Int := -260;   // Positioning request 3: Destination position
      Req4_Dest : Int := 0;   // Positioning request 4: Destination position
      Req1_Fwd : Bool := FALSE;   // Positioning request 1: Axis forward
      Req1_Bkw : Bool := FALSE;   // Positioning request 1: Axis backward
      Req1_Slow : Bool := FALSE;   // Positioning request 1: Axis slow speed
      Req1_Pos : Bool := FALSE;   // Positioning request 1: Axis in position
      Req2_Fwd : Bool := FALSE;   // Positioning request 2: Axis forward
      Req2_Bkw : Bool := FALSE;   // Positioning request 2: Axis backward
      Req2_Slow : Bool := FALSE;   // Positioning request 2: Axis slow speed
      Req2_Pos : Bool := FALSE;   // Positioning request 2: Axis in position
      Req3_Fwd : Bool := FALSE;   // Positioning request 3: Axis forward
      Req3_Bkw : Bool := FALSE;   // Positioning request 3: Axis backward
      Req3_Slow : Bool := FALSE;   // Positioning request 3: Axis slow speed
      Req3_Pos : Bool := FALSE;   // Positioning request 3: Axis in position
      Req4_Fwd : Bool := FALSE;   // Positioning request 4: Axis forward
      Req4_Bkw : Bool := FALSE;   // Positioning request 4: Axis backward
      Req4_Slow : Bool := FALSE;   // Positioning request 4: Axis slow speed
      Req4_Pos : Bool := FALSE;   // Positioning request 4: Axis in position
      Req5_Dest : Int := 0;   // Positioning request 5: Destination position
      Req6_Dest : Int := 0;   // Positioning request 6: Destination position
      Req7_Dest : Int := 0;   // Positioning request 7: Destination position
      Req8_Dest : Int := 0;   // Positioning request 8: Destination position
      Req5_Fwd : Bool := FALSE;   // Positioning request 5: Axis forward
      Req5_Bkw : Bool := FALSE;   // Positioning request 5: Axis backward
      Req5_Slow : Bool := FALSE;   // Positioning request 5: Axis slow speed
      Req5_Pos : Bool := FALSE;   // Positioning request 5: Axis in position
      Req6_Fwd : Bool := FALSE;   // Positioning request 6: Axis forward
      Req6_Bkw : Bool := FALSE;   // Positioning request 6: Axis backward
      Req6_Slow : Bool := FALSE;   // Positioning request 6: Axis slow speed
      Req6_Pos : Bool := FALSE;   // Positioning request 6: Axis in position
      Req7_Fwd : Bool := FALSE;   // Positioning request 7: Axis forward
      Req7_Bkw : Bool := FALSE;   // Positioning request 7: Axis backward
      Req7_Slow : Bool := FALSE;   // Positioning request 7: Axis slow speed
      Req7_Pos : Bool := FALSE;   // Positioning request 7: Axis in position
      Req8_Fwd : Bool := FALSE;   // Positioning request 8: Axis forward
      Req8_Bkw : Bool := FALSE;   // Positioning request 8: Axis backward
      Req8_Slow : Bool := FALSE;   // Positioning request 8: Axis slow speed
      Req8_Pos : Bool := FALSE;   // Positioning request 8: Axis in position
      dbw92 : Int := 2000;   // Time for arm rotation motor stop
      dbw94 : Int := 0;
      dbw96 : Int := 0;
      dbw98 : Int := 0;   // Time for conveyor motor stop
      dbw100 : Int := 0;   // Time for forward on arm rotation and conveyor inverter
      dbw102 : Int := 0;   // Time for backward on arm rotation and conveyor inverter
      dbw104 : Int := 0;
      dbw106 : Int := 0;
      dbw108 : Int := 0;
      dbw110 : Int := 0;
   END_VAR
BEGIN
END_DATA_BLOCK

DATA_BLOCK "DB06_Clamp"   // DB6
{ S7_Optimized_Access := 'FALSE' }
AUTHOR : Robopac
VERSION : 0.0
// stored: AutoNumber false, IsOnlyStoredInLoadMemory false, IsWriteProtectedInAS false
   VAR RETAIN
      dbx0_0 : Bool := FALSE;   // Welder contrast upward
      dbx0_1 : Bool := FALSE;   // Welder contrast downward
      dbx0_2 : Bool := FALSE;   // Welder unit upward
      dbx0_3 : Bool := FALSE;   // Welder unit downward
      dbx0_4 : Bool := FALSE;
      dbx0_5 : Bool := FALSE;   // Film clamp upward
      dbx0_6 : Bool := FALSE;   // Film clamp downward
      dbx0_7 : Bool := FALSE;   // Welder and cut unit forward
      dbx1_0 : Bool := FALSE;   // Welder and cut unit backward
      dbx1_1 : Bool := FALSE;
      dbx1_2 : Bool := FALSE;
      dbx1_3 : Bool := FALSE;
      dbx1_4 : Bool := FALSE;
      dbx1_5 : Bool := FALSE;
      dbx1_6 : Bool := FALSE;
      dbx1_7 : Bool := FALSE;
      dbx2_0 : Bool := FALSE;   // Welder contrast forward
      dbx2_1 : Bool := FALSE;   // Welder contrast backward
      dbx2_2 : Bool := FALSE;
      dbx2_3 : Bool := FALSE;
      dbx2_4 : Bool := FALSE;
      dbx2_5 : Bool := FALSE;
      dbx2_6 : Bool := FALSE;
      dbx2_7 : Bool := FALSE;
      dbb3 : Byte := 16#00;
      dbx4_0 : Bool := FALSE;   // Spool carrage upward to cover tail
      dbx4_1 : Bool := FALSE;   // Spool carrage downward after film tail covered
      dbx4_2 : Bool := FALSE;   // Spool carrage upward at the begining
      dbx4_3 : Bool := FALSE;   // Spool carriage height to pull film at begining
      dbx4_4 : Bool := FALSE;   // Support memory for revolution over welder contrast
      dbx4_5 : Bool := TRUE;   // Clamp carriage is not backward because wrapping cycle
      dbb5 : Byte := 16#00;
      dbw6 : Int := 0;
      dbw8 : Int := 0;
      dbw10 : Int := 500;   // Spool carriage height for film tail airblower
      dbw12 : Int := 0;   // Number of revolution to open clamp
      dbw14 : Int := 0;   // Spool carriage height for film tail wrapped
      dbw16 : Int := 200;   // Spool carriage height to enable revolution over clamp
      dbw18 : Int := 1942;
      dbw20 : Int := 0;
      dbw22 : Int := 0;
      dbw24 : Int := 0;
      dbw26 : Int := 0;
      dbw28 : Int := 0;
      dbw30 : Int := 0;
      dbw32 : Int := 0;
      dbw34 : Int := 0;
      dbw36 : Int := 0;
      dbw38 : Int := 0;
      dbw40 : Int := 0;   // Delay to open clamp (number of 100msec)
      dbw42 : Int := 0;   // Time to open clamp related to actual speed
      dbw44 : Int := 0;
      dbw46 : Int := 0;
      dbw48 : Int := 0;
   END_VAR
BEGIN
END_DATA_BLOCK

DATA_BLOCK "DB07_TopAux"   // DB7
{ S7_Optimized_Access := 'FALSE' }
AUTHOR : Robopac
VERSION : 0.0
// stored: AutoNumber false, IsOnlyStoredInLoadMemory false, IsWriteProtectedInAS false
   VAR RETAIN
      VB700 : Byte := 16#00;
      V701_0 : Bool := TRUE;   // Top film is wrapped
      V701_1 : Bool := FALSE;   // Support memory for top wrapped
      V701_2 : Bool := FALSE;
      V701_3 : Bool := FALSE;
      V701_4 : Bool := FALSE;
      V701_5 : Bool := FALSE;
      V701_6 : Bool := FALSE;
      V701_7 : Bool := FALSE;
   END_VAR
BEGIN
END_DATA_BLOCK

DATA_BLOCK "DB08_Prestretch"   // DB8
{ S7_Optimized_Access := 'FALSE' }
AUTHOR : Robopac
VERSION : 0.0
// stored: AutoNumber false, IsOnlyStoredInLoadMemory false, IsWriteProtectedInAS false
   VAR RETAIN
      dbx0_0 : Bool := FALSE;   // Support memory for prestretch PGSM or PGSA
      dbx0_1 : Bool := FALSE;
      dbx0_2 : Bool := FALSE;
      dbx0_3 : Bool := FALSE;
      dbx0_4 : Bool := FALSE;
      dbx0_5 : Bool := FALSE;
      dbx0_6 : Bool := FALSE;
      dbx0_7 : Bool := FALSE;
      dbw2 : Int := 0;
      dbw4 : Int := 0;
      dbw6 : Int := 0;
      dbw8 : Int := 0;
      dbw10 : Int := 0;   // Film provided for every revolution at max speed (mm per revolution)
      dbw12 : Int := 0;   // Film force value to apply to pallet (mm)
      dbd14 : DInt := 0;   // Support memory for film force to apply to pallet
      dbw18 : Int := 0;   // Film force value to apply to pallet (analog value)
      dbw20 : Int := 0;   // Film force value to apply to pallet (%)
      dbw22 : Int := 0;
      dbw24 : Int := 0;
      dbw26 : Int := 0;
      dbw28 : Int := 0;
      dbw30 : Int := 0;   // Gain for analog scaling
      dbw32 : Int := 200;   // Film prestretch value to apply to pallet
      dbd34 : DInt := 0;   // Support memory for film prestretch to apply to pallet
      dbw38 : Int := 102;   // Film prestretch value to apply to pallet (analog value)
      dbw40 : Int := 0;
      dbw42 : Int := 0;
      dbw44 : Int := 0;
      dbw46 : Int := 0;
      dbw48 : Int := 0;
      dbw50 : Int := 0;   // Support for film prestretch test
      dbw52 : Int := 0;   // Support for film prestretch test
      dbw54 : Int := 0;   // Film weight every mm of film (10^-5 g/mm)
      dbw56 : Int := 0;
      dbw58 : Int := 0;
      dbw60 : Int := 0;
   END_VAR
BEGIN
END_DATA_BLOCK

DATA_BLOCK "DB100_Display"   // DB100
{ S7_Optimized_Access := 'FALSE' }
VERSION : 0.1
// stored: AutoNumber false, IsOnlyStoredInLoadMemory false, IsWriteProtectedInAS false
   VAR RETAIN
      CELLA : Int := 15;   // CELLA (rosa)
      SETPOINT : UInt := 20;   // SETPOINT (rosso)
      PROP : Int := 0;   // PROPORZIONALE (verde)
      "INT" : Int := 0;   // INTEGRALE (giallo)
      FREQ_TIRO : Int := 0;   // U241
      FREQ_PRES : Int := 0;   // U261
   END_VAR
BEGIN
END_DATA_BLOCK

DATA_BLOCK "DB10_ExtConveyors"   // DB10
{ S7_Optimized_Access := 'FALSE' }
VERSION : 0.1
// stored: AutoNumber false, IsOnlyStoredInLoadMemory false, IsWriteProtectedInAS false
   VAR RETAIN
      V1000_0 : Bool := FALSE;
      V1000_1 : Bool := FALSE;
      V1000_2 : Bool := FALSE;
      V1000_3 : Bool := FALSE;
      V1000_4 : Bool := FALSE;
      V1000_5 : Bool := FALSE;
      V1000_6 : Bool := FALSE;
      V1000_7 : Bool := FALSE;
      V1001_0 : Bool := FALSE;
      V1001_1 : Bool := FALSE;
      V1001_2 : Bool := FALSE;
      V1001_3 : Bool := FALSE;
      V1001_4 : Bool := FALSE;
      V1001_5 : Bool := FALSE;
      V1001_6 : Bool := FALSE;
      V1001_7 : Bool := FALSE;
      Out_ConvPos1 : Bool := FALSE;   // Conveyor pos1 motor
      Out_ConvPos2 : Bool := FALSE;   // Conveyor pos2 motor
      Out_ConvPos3 : Bool := FALSE;   // Conveyor pos3 motor
      Out_ConvPos4 : Bool := FALSE;   // Conveyor pos4 motor
      Out_ConvPos5 : Bool := FALSE;   // Conveyor pos5 motor
      Out_ConvPos6 : Bool := FALSE;   // Conveyor pos6 motor
      Out_ConvPos7 : Bool := FALSE;   // Conveyor pos7 motor
      Out_ConvPos8 : Bool := FALSE;   // Conveyor pos8 motor
      Out_ConvPos1Rev : Bool := FALSE;   // Conveyor pos1 motor reverse
      Out_ConvPos2Rev : Bool := FALSE;   // Conveyor pos2 motor reverse
      Out_ConvPos3Rev : Bool := FALSE;   // Conveyor pos3 motor reverse
      Out_ConvPos4Rev : Bool := FALSE;   // Conveyor pos4 motor reverse
      V1003_4 : Bool := FALSE;
      V1003_5 : Bool := FALSE;
      V1003_6 : Bool := FALSE;
      V1003_7 : Bool := FALSE;
      VW1004 : Int := 0;
      Out_ConvPos1X2 : Bool := FALSE;   // Conveyor pos1 motor speed selection X2
      Out_ConvPos2X2 : Bool := FALSE;   // Conveyor pos2 motor speed selection X2
      Out_ConvPos3X2 : Bool := FALSE;   // Conveyor pos3 motor speed selection X2
      Out_ConvPos4X2 : Bool := FALSE;   // Conveyor pos4 motor speed selection X2
      V1006_4 : Bool := FALSE;
      V1006_5 : Bool := FALSE;
      V1006_6 : Bool := FALSE;
      V1006_7 : Bool := FALSE;
      Out_ConvPos2Upw : Bool := FALSE;   // Conveyor pos2 motor upward
      Out_ConvPos2Downw : Bool := FALSE;   // Conveyor pos2 downstroke valve command
      In_ConvPos2Up : Bool := TRUE;   // Conveyor pos2 up photocell NC
      In_ConvPos2Down : Bool := TRUE;   // Conveyor pos2 down photocell NC
      In_ConvPos2ExUp : Bool := TRUE;   // Conveyor pos2 up extrastroke switch NC
      In_ConvPos2Safety : Bool := TRUE;   // Conveyor pos2 down foot safety switch NC
      V1007_6 : Bool := FALSE;
      V1007_7 : Bool := FALSE;
   END_VAR
BEGIN
END_DATA_BLOCK

DATA_BLOCK "DB14_CutWireControl"   // DB14
{ S7_Optimized_Access := 'FALSE' }
VERSION : 0.1
// stored: AutoNumber false, IsOnlyStoredInLoadMemory false, IsWriteProtectedInAS false
   VAR RETAIN
      clean : Time := T#0MS;
      check : Time := T#0MS;
   END_VAR
BEGIN
END_DATA_BLOCK

DATA_BLOCK "DB20_DisplaySysdata"   // DB20
{ S7_Optimized_Access := 'FALSE' }
AUTHOR : Robopac
VERSION : 0.0
// stored: AutoNumber false, IsOnlyStoredInLoadMemory false, IsWriteProtectedInAS false
   VAR RETAIN
      dbd0 : DInt := 238;   // Step for encoder spool carriage movement (mm/100) (Display-Sysadata)
      dbw4 : Int := 6;   // Histeresys for spool carriage positioning (mm) (Display-Sysdata)
      dbw6 : Int := 50;   // Deceleration for spool carriage positioning (mm) (Display-Sysdata)
      dbw8 : Int := 50;   // Low speed for spool carriage movement (%) (Display-Sysdata)
      dbw10 : Int := 100;   // High speed for spool carriage movement (%) (Display-Sysdata)
      dbw12 : Int := 430;   // Spool height (mm) (Display-Sysdata)
      dbw14 : Int := 0;   // Spool carriage down position (mm) (Display-Sysadata)
      dbw16 : Int := 100;   // First step speed for spool carriage movement (%) (Display-Sysadata)
      dbw18 : Int := 240;   // Offset for ftc pallet height (mm) (Display-Sysdata)
      dbw20 : Int := 180;   // Pressure plate height (mm) (Display-Sysdata)
      dbw22 : Int := 7;   // Distance lifter up - conveyor (mm) (Display-Sysdata)
      dbw24 : Int := 0;   // Spool carriage height for film broken cycle (mm) (Display-Sysdata)
      dbw26 : Int := 50;   // Low speed angle to stop rotation (Display-Sysdata)
      dbw28 : Int := 1000;   // Jog1 speed for fast prestretch rool (Display-Sysadata)
      dbw30 : Int := 45;   // Offset for SCSP/2 (Display-Sysadata)
      dbw32 : Int := 78;
      dbw34 : Int := 1100;   // Arm rotation motor and gearbox type (Display-Sysdata)
      dbw36 : Int := 0;   // Delay for test cycle (Display-Sysdata)
      dbx38_0 : Bool := FALSE;   // Film ended or broken cycle included/excluded(1) (Display-Sysdata)
      dbx38_1 : Bool := FALSE;   // Conveyor encoder alarm included(0)/excluded (Display-Sysdata)
      dbx38_2 : Bool := FALSE;   // Test cycle included(1)/excluded (Display-Sysdata)
      dbx38_3 : Bool := FALSE;   // Top film ended or broken included(0)/excluded (Display-Sysdata)
      dbx38_4 : Bool := TRUE;   // Pallet height with pressure plate priority (Display-Sysdata)
      dbx38_5 : Bool := TRUE;   // Spool carriage upward during arm deceleration excluded/included(1) (Display-Sys
      dbx38_6 : Bool := FALSE;   // Pressure plate upward before(0)/after cut cycle (Display-Sysdata)
      dbx38_7 : Bool := FALSE;   // Bit stop pallet infeed (Display-Sysdata)
      dbx39_0 : Bool := FALSE;   // Timeout included/excluded(1) (Display-Sysdata)
      dbx39_1 : Bool := FALSE;   // Reverse cycle request from hmi (Display-Main page)
      dbx39_2 : Bool := FALSE;
      dbx39_3 : Bool := FALSE;
      dbx39_4 : Bool := FALSE;
      dbx39_5 : Bool := FALSE;
      dbx39_6 : Bool := TRUE;   // Top fast cycle
      dbx39_7 : Bool := FALSE;
      dbw40 : Int := 65;   // Spool carriage upward during arm deceleration (mm) (Display-Sysdata)
      dbw42 : Int := 1360;   // Step for infeed conveyor encoder (mm/100) (Display-Sysdata)
      dbw44 : Int := -210;   // Pulse offset for rotation encoder (Display-Sysdata)
      dbw46 : Int := 0;   // Pallet lenght for small pallet (Display-Sysdata)
      dbw48 : Int := 0;   // Decentering for pallet positioning (Display-Sysdata)
      dbw50 : Int := 500;   // Quote for airblower on (mm) (Display-Sysdata)
      dbw52 : Int := 0;   // Spool carriage up to cover film tail (Display-Sysdata)
      dbw54 : Int := 3000;   // Cutting time (Display-Sysdata)
      dbw56 : Int := 1500;   // MAX TIRO SU CELLA (kg) [ex SysdataTempoTwist]
      dbw58 : Int := 2400;   // Delay to open clamp (Display-Sysdata)
      dbw60 : Int := 0;   // Table rotation clampcut phase (°) (Display-Sysdata)
      dbw62 : Int := 200;   // Quote to open clamp (Display-Sysdata)
      dbw64 : Int := 0;   // Step for top carriage forward/backward (mm/100) (Display-Sysdata)
      dbw66 : Int := 1000;   // Step for top carriage upward/downward (mm/100) (Display-Sysdata)
      dbw68 : Int := 600;   // Deceleration for top carriage forward/backward (Display-Sysdata)
      dbw70 : Int := 1500;   // Top carriage up position (Display-Sysdata)
      dbw72 : Int := 0;   // Spool carriage position for top cycle (Display-Sysdata)
      dbw74 : Int := 0;   // Delay for spool carriage downward during top cycle (Display-Sysdata)
      dbw76 : Int := 0;   // Tabke rotation load phase (°) (Display-Sysdata)
      dbw78 : Int := 0;   // Table rotation unload phase (°) (Display-Sysdata)
      dbd80 : DInt := 5627;   // Step for encoder table rotation movement (°/p) (Display-Sysdata)
      dbw84 : Int := 18;   // Histeresys for table rotation positioning (°) (Display-Sysdata)
      dbw86 : Int := 2100;   // Deceleration for table rotation positioning (Hz/sec) (Display-Sysdata)
      dbw88 : Int := 10;   // Low speed for table rotation movement (%) (Display-Sysdata)
      dbw90 : Int := 100;   // High speed for table rotation movement (%) (Display-Sysdata)
      dbw92 : Int := 1800;   // Delay to stop top carriage forward for top film broken
      dbw94 : Int := 1000;   // Delay for top pallet height reading photocell (fast cycle)
      dbw96 : Int := 60;
      dbw98 : Int := 20;
   END_VAR
BEGIN
END_DATA_BLOCK

DATA_BLOCK "DB215_ProgramData"   // DB215
TITLE = Program Data
{ S7_Optimized_Access := 'FALSE' }
VERSION : 0.1
// stored: AutoNumber false, IsOnlyStoredInLoadMemory false, IsWriteProtectedInAS false
   VAR RETAIN
      State_Initialization : UInt := 0;
      State_Setup : UInt := 0;
      InverterFault : Bool := FALSE;   // Inverter Fault (F) - Anomalia
      InverterAlarm : Bool := FALSE;   // Inverter Alarm (A) - Avviso
      Keylock : Bool := FALSE;   // Blocco tasti per utente
      ActiveRecipeMLC : Bool := FALSE;   // Multi-Level Control per la ricetta attiva
      Keylock2 : Bool := FALSE;   // Blocco tasti (StateAuto opp. blocco)
      RecipeModified : Bool := FALSE;
      RecipeSave : Bool := FALSE;
      LoadCellConst : Bool := TRUE;   // valore cella costante
      spare_5 : Bool := FALSE;
      spare_6 : Bool := FALSE;
      spare_7 : Bool := FALSE;
      spare_8 : Bool := FALSE;
      spare_9 : Bool := FALSE;
      spare_10 : Bool := FALSE;
      spare_11 : Bool := FALSE;
      spare_12 : Bool := FALSE;
      Offset_Pulses : Int := 0;   // NOT_USED
      Altimeter_Pulses : Int := 442;
      PhotDelay_Pulses : Int := 40;
      Reinforce_Pulses : Int := 0;
      TopFall_Pulses : Int := 134;
      ManRotStep : UInt := 0;
      RotSpeed : Int := 1770;
      CarSpeedUp : Int := 1396;
      CarSpeedDw : Int := 1396;
      Offset_cella : Int := 240;
      EncCarrDir : Int := -1;   // Direzione petalo carrello (1=av;-1=ind)
      EncCarrMax : Int := 603;   // Max altezza carrello (encoder)
      TiroObiettivo : UInt := 0;   // Tiro obiettivo (da chiamata FC300)
      ContaImpulsi : Int := 0;   // Contatore impulsi 20ms (OB30)
      MLC_HeightPulses : Int := 0;   // MLC_Height_Pulses
      MLC_Rounds : Int := 0;   // MLC_rounds
      LoadCellVal_1 : Int := 227;   // valore cella 1
      LoadCellVal_2 : Int := 227;   // valore cella 2
      PropArmMax : Int := 0;   // Costante proporzionalità corrisp. max freq. braccio
      PropCarrMax : Int := 0;   // Costante proporzionalità corrisp. max freq. carrello
      ValOffsetCella : Int := 10;   // Valore per offset cella durante il reset
      RoundTime : UInt := 4000;
      LastRoundTime : UInt := 2000;
      ReinforceTime : UInt := 0;   // [NOT USED]
      pTiro : Array[0..10] of UInt;
      iTiro : Array[0..10] of UInt;
   END_VAR
BEGIN
   pTiro[0] := 70;
   pTiro[1] := 60;
   pTiro[2] := 50;
   pTiro[3] := 45;
   pTiro[4] := 40;
   pTiro[5] := 35;
   pTiro[6] := 30;
   pTiro[7] := 25;
   pTiro[8..10] := 20;
   iTiro[0] := 70;
   iTiro[1] := 60;
   iTiro[2] := 50;
   iTiro[3] := 45;
   iTiro[4] := 40;
   iTiro[5] := 35;
   iTiro[6] := 30;
   iTiro[7] := 25;
   iTiro[8..10] := 20;
END_DATA_BLOCK

DATA_BLOCK "DB22_DisplayData"   // DB22
{ S7_Optimized_Access := 'FALSE' }
AUTHOR : Robopac
VERSION : 0.0
// stored: AutoNumber false, IsOnlyStoredInLoadMemory false, IsWriteProtectedInAS false
   VAR RETAIN
      dbx0_0 : Bool := FALSE;   // Technoplat manual(Display): Table rotation forward
      dbx0_1 : Bool := FALSE;   // Technoplat manual(Display): Spool carriage upward
      dbx0_2 : Bool := FALSE;   // Technoplat manual(Display): Spool carriage downward
      dbx0_3 : Bool := FALSE;   // Technoplat manual(Display): Pressure plate upward/downward
      dbx0_4 : Bool := FALSE;   // Technoplat manual(Display): Pallet lifter upward/downward
      dbx0_5 : Bool := FALSE;   // Technoplat manual(Display): Rope unit open/close
      dbx0_6 : Bool := FALSE;   // Technoplat manual(Display): Prestretch
      dbx0_7 : Bool := FALSE;   // Technoplat manual(Display): Spool carriage to film broken position
      dbx1_0 : Bool := FALSE;   // Clamp manual(Display): Clamp upward/downward
      dbx1_1 : Bool := FALSE;   // Clamp manual(Display): Welder unit upward/downward
      dbx1_2 : Bool := FALSE;   // Clamp manual(Display): Welder contrast upward/downward
      dbx1_3 : Bool := FALSE;   // Clamp manual(Display): Clamp carriage forward/backward
      dbx1_4 : Bool := FALSE;   // Clamp manual(Display): Clamp open/close
      dbx1_5 : Bool := FALSE;   // Clamp manual(Display): Cut and welder arm forward/backward
      dbx1_6 : Bool := FALSE;   // Clamp manual(Display): Welder unit forward/backward
      dbx1_7 : Bool := FALSE;   // Clamp manual(Display):
      dbx2_0 : Bool := FALSE;   // Top manual(Display): Top carriage upward
      dbx2_1 : Bool := FALSE;   // Top manual(Display): Top carriage downward
      dbx2_2 : Bool := FALSE;   // Top manual(Display): Top carriage forward
      dbx2_3 : Bool := FALSE;   // Top manual(Display): Top carriage backward
      dbx2_4 : Bool := FALSE;   // Top manual(Display): Opening/closing clamp to pull top film
      dbx2_5 : Bool := FALSE;   // Top manual(Display): Opening/closing clamp to block top film
      dbx2_6 : Bool := FALSE;   // Top manual(Display): Top film cutter forward/backward
      dbx2_7 : Bool := FALSE;   // Top manual(Display): Arm rotation to phase 2 sensor for top
      dbx3_0 : Bool := FALSE;   // Technoplat manual (Display): Rotation to unload
      dbx3_1 : Bool := FALSE;   // Technoplat manual (Display): Rotation to 0
      dbx3_2 : Bool := FALSE;   // Technoplat manual (Display): Rotation to load
      dbx3_3 : Bool := FALSE;
      dbx3_4 : Bool := FALSE;   // Technoplat manual(Display): Rope unit lower open/close
      dbx3_5 : Bool := FALSE;
      dbx3_6 : Bool := FALSE;
      dbx3_7 : Bool := FALSE;
      dbx4_0 : Bool := FALSE;   // Conveyor manual(Display): CMD PRESSED
      dbx4_1 : Bool := FALSE;   // Conveyor manual(Display): Load CM [p18]
      dbx4_2 : Bool := FALSE;   // Conveyor manual(Display): Unload CM [p18]
      dbx4_3 : Bool := FALSE;   // Conveyor manual(Display): RESET ENCODER
      dbx4_4 : Bool := FALSE;   // Conveyor manual(Display): Load CM [Sysdata]
      dbx4_5 : Bool := FALSE;   // Conveyor manual(Display): [not used]
      dbx4_6 : Bool := FALSE;   // Conveyor manual(Display): CM backward slow
      dbx4_7 : Bool := FALSE;   // Conveyor manual(Display): CM forward slow
      dbb5 : Byte := 16#09;   // Conveyor manual operation
      dbx6_0 : Bool := FALSE;   // Manual Signal(Display): Pallet ready in infeed (Input)
      dbx6_1 : Bool := FALSE;   // Manual Signal(Display): Ready to receive pallet infeed (Output)
      dbx6_2 : Bool := FALSE;   // Manual Signal(Display): End of transfer pallet infeed (Output)
      dbx6_3 : Bool := FALSE;   // Manual Signal(Display): Pallet ready in outfeed (Output)
      dbx6_4 : Bool := FALSE;   // Manual Signal(Display): Ready to receive pallet outfeed (Input)
      dbx6_5 : Bool := FALSE;   // Manual Signal(Display): End of transfer pallet outfeed (Input)
      dbx6_6 : Bool := FALSE;   // Manual Signal(Display): Start wrapping signal (Input)
      dbx6_7 : Bool := FALSE;   // Manual Signal(Display): Customer conveyor stopped signal (Input)
      dbx7_0 : Bool := FALSE;   // Manual Signal(Display): Machine in position signal (Output)
      dbx7_1 : Bool := FALSE;   // Manual Signal(Display): Wrapp ended signal (Output)
      dbx7_2 : Bool := FALSE;   // Manual Signal(Display): Pallet in position for label
      dbx7_3 : Bool := TRUE;   // Manual Signal(Display): Label arm in position for pallet transfer
      dbx7_4 : Bool := FALSE;   // Manual Signal(Display): Label cycle ended
      dbx7_5 : Bool := FALSE;   // Manual Signal(Display): Label fault
      dbx7_6 : Bool := FALSE;
      dbx7_7 : Bool := FALSE;
      dbw8 : Int := 0;
      dbw10 : Int := 0;
      dbw12 : Int := 0;
      dbx14_0 : Bool := FALSE;   // Technoplat manual(Program): Table rotation forward
      dbx14_1 : Bool := FALSE;   // Technoplat manual(Program): Spool carriage upward
      dbx14_2 : Bool := FALSE;   // Technoplat manual(Program): Spool carriage downward
      dbx14_3 : Bool := FALSE;   // Technoplat manual(Program): Pressure plate downward
      dbx14_4 : Bool := FALSE;   // Technoplat manual(Program): Pressure plate upward
      dbx14_5 : Bool := FALSE;   // Technoplat manual(Program): Pallet lifter upward
      dbx14_6 : Bool := FALSE;   // Technoplat manual(Program): Pallet lifter downward
      dbx14_7 : Bool := FALSE;   // Technoplat manual(Program): Rope unit closing
      dbx15_0 : Bool := FALSE;   // Technoplat manual(Program): Rope unit opening
      dbx15_1 : Bool := FALSE;   // Technoplat manual(Program): Prestretch
      dbx15_2 : Bool := FALSE;   // Technoplat manual(Program): Spool carriage to film broken position
      dbx15_3 : Bool := FALSE;   // Technoplat manual(Program): Rope unit Lower closing
      dbx15_4 : Bool := FALSE;   // Technoplat manual(Program): Rope unit Lower opening
      dbx15_5 : Bool := FALSE;   // Technoplat manual(Program): CM Backward slow
      dbx15_6 : Bool := FALSE;   // Technoplat manual(Program): CM Forward slow
      dbx15_7 : Bool := FALSE;   // Technoplat manual(Program):
      dbx16_0 : Bool := FALSE;   // Clamp manual(Program): Clamp upward
      dbx16_1 : Bool := FALSE;   // Clamp manual(Program): Clamp downward
      dbx16_2 : Bool := FALSE;   // Clamp manual(Program): Welder unit upward
      dbx16_3 : Bool := FALSE;   // Clamp manual(Program): Welder unit downward
      dbx16_4 : Bool := FALSE;   // Clamp manual(Program): Welder contrast upward
      dbx16_5 : Bool := FALSE;   // Clamp manual(Program): Welder contrast downward
      dbx16_6 : Bool := FALSE;   // Clamp manual(Program): Clamp carriage forward
      dbx16_7 : Bool := FALSE;   // Clamp manual(Program): Clamp carriage backward
      dbx17_0 : Bool := FALSE;   // Clamp manual(Program): Clamp open
      dbx17_1 : Bool := FALSE;   // Clamp manual(Program): Clamp close
      dbx17_2 : Bool := FALSE;   // Clamp manual(Program): Cut and welder arm forward
      dbx17_3 : Bool := FALSE;   // Clamp manual(Program): Cut and welder arm backward
      dbx17_4 : Bool := FALSE;   // Clamp manual(Program): Welder unit forward
      dbx17_5 : Bool := FALSE;   // Clamp manual(Program): Welder unit backward
      dbx17_6 : Bool := FALSE;   // Clamp manual(Program):
      dbx17_7 : Bool := FALSE;   // Clamp manual(Program):
      dbx18_0 : Bool := FALSE;   // Top manual(Program): Top carriage upward
      dbx18_1 : Bool := FALSE;   // Top manual(Program): Top carriage downward
      dbx18_2 : Bool := FALSE;   // Top manual(Program): Top carriage forward
      dbx18_3 : Bool := FALSE;   // Top manual(Program): Top carriage backward
      dbx18_4 : Bool := FALSE;   // Top manual(Program): Opening clamp to pull top film
      dbx18_5 : Bool := FALSE;   // Top manual(Program): Closing clamp to pull top film
      dbx18_6 : Bool := FALSE;   // Top manual(Program): Opening clamp to block top film
      dbx18_7 : Bool := FALSE;   // Top manual(Program): Closing clamp to block top film
      dbx19_0 : Bool := FALSE;   // Top manual(Program): Top film cutter forward/backward
      dbx19_1 : Bool := FALSE;   // Top manual(Program): Arm rotation to phase 2 sensor for top
      dbx19_2 : Bool := FALSE;   // Technoplat manual(Program): Rotation to unload
      dbx19_3 : Bool := FALSE;   // Technoplat manual(Program): Rotation to 0
      dbx19_4 : Bool := FALSE;   // Technoplat manual(Program): Rotation to load
      dbx19_5 : Bool := FALSE;   // Top manual(Program):
      dbx19_6 : Bool := FALSE;   // Top manual(Program):
      dbx19_7 : Bool := FALSE;   // Top manual(Program):
      dbx20_0 : Bool := FALSE;   // Conveyor manual(Program): Load CM
      dbx20_1 : Bool := FALSE;   // Conveyor manual(Program): Unload CM
      dbx20_2 : Bool := FALSE;   // Conveyor manual(Program): CM backward
      dbx20_3 : Bool := FALSE;   // Conveyor manual(Program): Pos.1
      dbx20_4 : Bool := FALSE;   // Conveyor manual(Program): Pos.2
      dbx20_5 : Bool := FALSE;   // Conveyor manual(Program): Pos.3
      dbx20_6 : Bool := FALSE;   // Conveyor manual(Program): Pos.4
      dbx20_7 : Bool := FALSE;   // Conveyor manual(Program): Pos.5
      dbx21_0 : Bool := FALSE;   // Conveyor manual(Program): Pos.6
      dbx21_1 : Bool := FALSE;   // Conveyor manual(Program): Pos.7
      dbx21_2 : Bool := FALSE;   // Conveyor manual(Program): Pos.8
      dbx21_3 : Bool := FALSE;   // Conveyor manual(Program):
      dbx21_4 : Bool := FALSE;   // Conveyor manual(Program):
      dbx21_5 : Bool := FALSE;   // Conveyor manual(Program):
      dbx21_6 : Bool := FALSE;   // Conveyor manual(Program):
      dbx21_7 : Bool := FALSE;   // Conveyor manual(Program):
      dbx22_0 : Bool := FALSE;   // Manual Signal(Program): Pallet ready in infeed (Input)
      dbx22_1 : Bool := FALSE;   // Manual Signal(Program): Ready to receive pallet infeed (Output)
      dbx22_2 : Bool := FALSE;   // Manual Signal(Program): End of transfer pallet infeed (Output)
      dbx22_3 : Bool := FALSE;   // Manual Signal(Program): Pallet ready in outfeed (Output)
      dbx22_4 : Bool := FALSE;   // Manual Signal(Program): Ready to receive pallet outfeed (Input)
      dbx22_5 : Bool := FALSE;   // Manual Signal(Program): End of transfer pallet outfeed (Input)
      dbx22_6 : Bool := FALSE;   // Manual Signal(Program): Start wrapping (Input)
      dbx22_7 : Bool := FALSE;   // Manual Signal(Program): Customer conveyor stopped (Input)
      dbx23_0 : Bool := FALSE;   // Manual Signal(Program): Machine in position (Output)
      dbx23_1 : Bool := FALSE;   // Manual Signal(Program): Wrapp ended (Output)
      dbx23_2 : Bool := FALSE;   // Manual Signal(Program): Pallet ready for label
      dbx23_3 : Bool := TRUE;   // Manual Signal(Program): Label arm in position for pallet transfer
      dbx23_4 : Bool := FALSE;   // Manual Signal(Program): Label cycle ended
      dbx23_5 : Bool := FALSE;   // Manual Signal(Program): Label fault
      dbx23_6 : Bool := FALSE;
      dbx23_7 : Bool := FALSE;
      dbw24 : Int := 0;
      dbw26 : Int := 0;
      dbw28 : Int := 0;
      dbw30 : Int := 0;
      dbx32_0 : Bool := TRUE;   // Manual(Toggle bit): Pressure plate upward/downward (Technplat)
      dbx32_1 : Bool := TRUE;   // Manual(Toggle bit): Pallet lifter upward/downward (Technplat)
      dbx32_2 : Bool := FALSE;   // Manual(Toggle bit): Clamp upward/downward (Clamp)
      dbx32_3 : Bool := FALSE;   // Manual(Toggle bit): Welder unit upward/downward (Clamp)
      dbx32_4 : Bool := TRUE;   // Manual(Toggle bit): Welder contrast upward/downward (Clamp)
      dbx32_5 : Bool := FALSE;   // Manual(Toggle bit): Rope unit open/close (Technplat)
      dbx32_6 : Bool := FALSE;   // Manual(Toggle bit): Clamp open/close (Clamp)
      dbx32_7 : Bool := FALSE;   // Manual(Toggle bit): Cut and welder arm forward/backward (Clamp)
      dbx33_0 : Bool := TRUE;   // Manual(Toggle bit): Opening/closing clamp to pull top film (Top)
      dbx33_1 : Bool := TRUE;   // Manual(Toggle bit): Opening/closing clamp to block top film (Top)
      dbx33_2 : Bool := TRUE;   // Manual(Toggle bit): Welder unit forward/backward (Clamp)
      dbx33_3 : Bool := FALSE;   // Manual(Toggle bit): Clamp carriage forward/backward (Clamp)
      dbx33_4 : Bool := FALSE;   // Manual(Toggle bit): Rope unit lower open/close (Technplat)
      dbx33_5 : Bool := FALSE;   // Manual(Toggle bit):
      dbx33_6 : Bool := FALSE;   // Manual(Toggle bit):
      dbx33_7 : Bool := FALSE;   // Manual(Toggle bit):
      dbw34 : Int := 0;
      dbw36 : Int := 0;
      dbx38_0 : Bool := FALSE;   // Diagnostic signal conveyor: Pallet ready in infeed (input)
      dbx38_1 : Bool := TRUE;   // Diagnostic signal conveyor: Ready to receive pallet infeed (Output)
      dbx38_2 : Bool := FALSE;   // Diagnostic signal conveyor: End of transfer pallet infeed (Output)
      dbx38_3 : Bool := FALSE;   // Diagnostic signal conveyor: Ready to receive pallet in outfeed (Input)
      dbx38_4 : Bool := FALSE;   // Diagnostic signal conveyor: End of transfer pallet outfeed (Input)
      dbx38_5 : Bool := FALSE;   // Diagnostic signal conveyor: Pallet ready in outfeed (Output)
      dbx38_6 : Bool := FALSE;   // Diagnostic signal conveyor: Start wrapping (Input)
      dbx38_7 : Bool := FALSE;   // Diagnostic signal conveyor: Customer conveyor stopped (Input)
      dbx39_0 : Bool := FALSE;   // Diagnostic signal conveyor: Machine in position (Output)
      dbx39_1 : Bool := FALSE;   // Diagnostic signal conveyor: Wrapp ended (Output)
      dbx39_2 : Bool := FALSE;   // Diagnostic signal conveyor: Pallet ready for label
      dbx39_3 : Bool := TRUE;   // Diagnostic signal conveyor: Label arm in position for pallet transit
      dbx39_4 : Bool := FALSE;   // Diagnostic signal conveyor: Label cycle ended
      dbx39_5 : Bool := FALSE;   // Diagnostic signal conveyor: Label fault
      dbw40 : Int := 1;   // Machine status
      dbd42 : DInt := 4;   // Worked hours
      dbd46 : DInt := 95;   // Partial counter for wrapped pallet
      dbd50 : DInt := 163;   // Counter for wrapped pallet
      dbd54 : DInt := 0;
      dbw58 : Int := 21;   // Seconds for worked hours counter
      dbw60 : Int := 36;   // Minutes for worked hours counter
      dbw62 : Int := 0;   // Arm rotation speed (rpm)
      dbw64 : Int := 0;   // Arm rotation speed (rpm)
      dbw66 : Int := 15;   // Number of revolution done on last pallet
      dbw68 : Int := 777;   // Wrapping cycle time
      dbw70 : Int := 22482;   // Wrapping cycle + pallet transfer time
      dbw72 : Int := 10;   // Pallet per hour (Productivity)
      dbw74 : Int := 0;   // Film weight every wrapping cycle (g*10)
      dbw76 : Int := 0;   // Film force for film weight value
      dbw78 : Int := 0;   // Film prestretch for film weight value
      dbw80 : Int := 0;
      dbw82 : Int := 0;
      dbw84 : Int := 0;
      dbw86 : Int := 0;
      dbw88 : Int := 0;
      dbw90 : Int := 0;
      dbw92 : Int := 0;
      dbw94 : Int := 0;
      dbw96 : Int := 0;
      dbw98 : Int := 0;
   END_VAR
BEGIN
END_DATA_BLOCK

DATA_BLOCK "DB235_Program15"   // DB235
{ S7_Optimized_Access := 'FALSE' }
AUTHOR : Robopac
VERSION : 0.0
// stored: AutoNumber false, IsOnlyStoredInLoadMemory false, IsWriteProtectedInAS false
   VAR RETAIN
      Program15 { S7_SetPoint := 'True'} : "DatiProgramma";
   END_VAR
BEGIN
   Program15.Wrapping := TRUE;
   Program15.TopLenght := 500;
   Program15.TopRelease := 0;
   Program15.TopDown := 0;
   Program15.Top := 4;
   Program15.PressurePTime := 0;
   Program15.LifterTime := 0;
   Program15.RevOverContrast := 1;
   Program15.RopeEndCycle := 16#02;
   Program15.Spare4 := 16#01;
   Program15.RopeTime := 1500;
   Program15.RevOverClamp := 1;
   Program15.FilmForceFinalRev := 10;
   Program15.FilmPrestretchFinalRev := 100;
   Program15.ArmSpeed := 100;
   Program15.CarriageDown4Top := 500;
   Program15.TopDownTime := 1500;
   Program15.LapsUnderTop := 0;
   Program15.Spare6 := 0;
   Program15.Spare7 := 0;
   Program15.Spare8 := 0;
   Program15.Spare9 := 0;
   Program15.Spare10 := 0;
   Program15.Spare11 := 0;
   Program15.Spare12 := 0;
   Program15.Overlap0_1 := 0;
   Program15.Height1 := 130;
   Program15.Landmark1 := FALSE;
   Program15.Lifter1 := FALSE;
   Program15.SpareBit1H1 := FALSE;
   Program15.Airblower1 := TRUE;
   Program15.NextStep1 := TRUE;
   Program15.PressureP1 := TRUE;
   Program15.SpareByte2H1 := 16#00;
   Program15.Revolution1 := 1;
   Program15.RopeUnit1_1 := 16#01;
   Program15.RopeUnit1_2 := 16#01;
   Program15.FilmForce1 := 5;
   Program15.FilmPrestretch1 := 200;
   Program15.Spare3H1 := 0;
   Program15.Spare49 := 0;
   Program15.Spare50 := 0;
   Program15.Spare51 := 0;
   Program15.Spare52 := 0;
   Program15.Spare53 := 0;
   Program15.Overlap1_2 := 0;
   Program15.Height2 := 50;
   Program15.Landmark2 := FALSE;
   Program15.Lifter2 := FALSE;
   Program15.SpareBit1H2 := FALSE;
   Program15.Airblower2 := TRUE;
   Program15.NextStep2 := TRUE;
   Program15.PressureP2 := TRUE;
   Program15.SpareByte2H2 := 16#00;
   Program15.Revolution2 := 1;
   Program15.RopeUnit2_1 := 16#01;
   Program15.RopeUnit2_2 := 16#01;
   Program15.FilmForce2 := 20;
   Program15.FilmPrestretch2 := 200;
   Program15.Spare3H2 := 0;
   Program15.Spare54 := 0;
   Program15.Spare55 := 0;
   Program15.Spare56 := 0;
   Program15.Spare57 := 0;
   Program15.Spare58 := 0;
   Program15.Overlap2_3 := 100;
   Program15.Height3 := -50;
   Program15.Landmark3 := TRUE;
   Program15.Lifter3 := FALSE;
   Program15.SpareBit1H3 := FALSE;
   Program15.Airblower3 := TRUE;
   Program15.NextStep3 := TRUE;
   Program15.PressureP3 := TRUE;
   Program15.SpareByte2H3 := 16#00;
   Program15.Revolution3 := 2;
   Program15.RopeUnit3_1 := 16#01;
   Program15.RopeUnit3_2 := 16#01;
   Program15.FilmForce3 := 30;
   Program15.FilmPrestretch3 := 200;
   Program15.Spare3H3 := 0;
   Program15.Spare59 := 0;
   Program15.Spare60 := 0;
   Program15.Spare61 := 380;
   Program15.Spare62 := 2800;
   Program15.Spare63 := 0;
   Program15.Overlap3_4 := 100;
   Program15.Height4 := 100;
   Program15.Landmark4 := FALSE;
   Program15.Lifter4 := FALSE;
   Program15.SpareBit1H4 := FALSE;
   Program15.Airblower4 := TRUE;
   Program15.NextStep4 := TRUE;
   Program15.PressureP4 := TRUE;
   Program15.SpareByte2H4 := 16#00;
   Program15.Revolution4 := 3;
   Program15.RopeUnit4_1 := 16#02;
   Program15.RopeUnit4_2 := 16#02;
   Program15.FilmForce4 := 30;
   Program15.FilmPrestretch4 := 200;
   Program15.Spare3H4 := 0;
   Program15.Spare64 := 0;
   Program15.Spare65 := 0;
   Program15.Spare66 := 0;
   Program15.Spare67 := 0;
   Program15.Spare68 := 0;
   Program15.Overlap4_5 := 0;
   Program15.Height5 := 50;
   Program15.Landmark5 := FALSE;
   Program15.Lifter5 := FALSE;
   Program15.SpareBit1H5 := FALSE;
   Program15.Airblower5 := TRUE;
   Program15.NextStep5 := FALSE;
   Program15.PressureP5 := FALSE;
   Program15.SpareByte2H5 := 16#00;
   Program15.Revolution5 := 1;
   Program15.RopeUnit5_1 := 16#01;
   Program15.RopeUnit5_2 := 16#01;
   Program15.FilmForce5 := 30;
   Program15.FilmPrestretch5 := 200;
   Program15.Spare3H5 := 0;
   Program15.Spare69 := 0;
   Program15.Spare70 := 0;
   Program15.Spare71 := 0;
   Program15.Spare72 := 0;
   Program15.Spare73 := 0;
   Program15.Overlap5_6 := 100;
   Program15.Height6 := 50;
   Program15.Landmark6 := FALSE;
   Program15.Lifter6 := FALSE;
   Program15.SpareBit1H6 := FALSE;
   Program15.Airblower6 := TRUE;
   Program15.NextStep6 := FALSE;
   Program15.PressureP6 := FALSE;
   Program15.SpareByte2H6 := 16#00;
   Program15.Revolution6 := 2;
   Program15.RopeUnit6_1 := 16#02;
   Program15.RopeUnit6_2 := 16#01;
   Program15.FilmForce6 := 20;
   Program15.FilmPrestretch6 := 200;
   Program15.Spare3H6 := 0;
   Program15.Spare74 := 0;
   Program15.Spare75 := 0;
   Program15.Spare76 := 0;
   Program15.Spare77 := 0;
   Program15.Spare78 := 0;
   Program15.Overlap6_7 := 0;
   Program15.Height7 := 0;
   Program15.Landmark7 := FALSE;
   Program15.Lifter7 := FALSE;
   Program15.SpareBit1H7 := FALSE;
   Program15.Airblower7 := FALSE;
   Program15.NextStep7 := TRUE;
   Program15.PressureP7 := FALSE;
   Program15.SpareByte2H7 := 16#00;
   Program15.Revolution7 := 1;
   Program15.RopeUnit7_1 := 16#01;
   Program15.RopeUnit7_2 := 16#01;
   Program15.FilmForce7 := 0;
   Program15.FilmPrestretch7 := 100;
   Program15.Spare3H7 := 0;
   Program15.Spare79 := 0;
   Program15.Spare80 := 0;
   Program15.Spare81 := 0;
   Program15.Spare82 := 0;
   Program15.Spare83 := 0;
   Program15.Overlap7_8 := 0;
   Program15.Height8 := 0;
   Program15.Landmark8 := FALSE;
   Program15.Lifter8 := FALSE;
   Program15.SpareBit1H8 := FALSE;
   Program15.Airblower8 := FALSE;
   Program15.NextStep8 := TRUE;
   Program15.PressureP8 := FALSE;
   Program15.SpareByte2H8 := 16#00;
   Program15.Revolution8 := 1;
   Program15.RopeUnit8_1 := 16#01;
   Program15.RopeUnit8_2 := 16#01;
   Program15.FilmForce8 := 0;
   Program15.FilmPrestretch8 := 100;
   Program15.Spare3H8 := 0;
   Program15.Spare84 := 0;
   Program15.Spare85 := 0;
   Program15.Spare86 := 0;
   Program15.Spare87 := 0;
   Program15.Spare88 := 0;
   Program15.Overlap8_9 := 0;
   Program15.Height9 := 0;
   Program15.Landmark9 := FALSE;
   Program15.Lifter9 := FALSE;
   Program15.SpareBit1H9 := FALSE;
   Program15.Airblower9 := FALSE;
   Program15.NextStep9 := TRUE;
   Program15.PressureP9 := FALSE;
   Program15.SpareByte2H9 := 16#00;
   Program15.Revolution9 := 1;
   Program15.RopeUnit9_1 := 16#01;
   Program15.RopeUnit9_2 := 16#01;
   Program15.FilmForce9 := 0;
   Program15.FilmPrestretch9 := 100;
   Program15.Spare3H9 := 0;
   Program15.Spare89 := 0;
   Program15.Spare90 := 0;
   Program15.Spare91 := 0;
   Program15.Spare92 := 0;
   Program15.Spare93 := 0;
   Program15.Overlap9_10 := 0;
   Program15.Height10 := 0;
   Program15.Landmark10 := FALSE;
   Program15.Lifter10 := FALSE;
   Program15.SpareBit1H10 := FALSE;
   Program15.Airblower10 := FALSE;
   Program15.NextStep10 := FALSE;
   Program15.PressureP10 := FALSE;
   Program15.SpareByte2H10 := 16#00;
   Program15.Revolution10 := 1;
   Program15.RopeUnit10_1 := 16#01;
   Program15.RopeUnit10_2 := 16#01;
   Program15.FilmForce10 := 0;
   Program15.FilmPrestretch10 := 100;
   Program15.Spare3H10 := 0;
   Program15.Spare94 := 0;
   Program15.Spare95 := 0;
   Program15.Spare96 := 0;
   Program15.Spare97 := 0;
   Program15.Spare98 := 0;
   Program15.Overlap10_11 := 0;
   Program15.Height11 := 0;
   Program15.Landmark11 := FALSE;
   Program15.Lifter11 := FALSE;
   Program15.SpareBit1H11 := FALSE;
   Program15.Airblower11 := FALSE;
   Program15.NextStep11 := TRUE;
   Program15.PressureP11 := FALSE;
   Program15.SpareByte2H11 := 16#00;
   Program15.Revolution11 := 1;
   Program15.RopeUnit11_1 := 16#01;
   Program15.RopeUnit11_2 := 16#01;
   Program15.FilmForce11 := 0;
   Program15.FilmPrestretch11 := 100;
   Program15.Spare3H11 := 0;
   Program15.Spare99 := 0;
   Program15.Spare100 := 0;
   Program15.Spare101 := 0;
   Program15.Spare102 := 0;
   Program15.Spare103 := 0;
   Program15.Overlap11_12 := 0;
   Program15.Height12 := 0;
   Program15.Landmark12 := FALSE;
   Program15.Lifter12 := FALSE;
   Program15.SpareBit1H12 := FALSE;
   Program15.Airblower12 := FALSE;
   Program15.NextStep12 := FALSE;
   Program15.PressureP12 := FALSE;
   Program15.SpareByte2H12 := 16#00;
   Program15.Revolution12 := 1;
   Program15.RopeUnit12_1 := 16#01;
   Program15.RopeUnit12_2 := 16#01;
   Program15.FilmForce12 := 0;
   Program15.FilmPrestretch12 := 100;
   Program15.Spare3H12 := 0;
   Program15.Spare104 := 0;
   Program15.Spare105 := 0;
   Program15.Spare106 := 0;
   Program15.Spare107 := 0;
   Program15.Spare108 := 0;
END_DATA_BLOCK

DATA_BLOCK "DB23_AlarmProgram"   // DB23
{ S7_Optimized_Access := 'FALSE' }
AUTHOR : Robopac
VERSION : 0.0
// stored: AutoNumber false, IsOnlyStoredInLoadMemory false, IsWriteProtectedInAS false
   VAR RETAIN
      dbx0_0 : Bool := FALSE;   // Alarm 1: Pressure switch (Technoplat)
      dbx0_1 : Bool := FALSE;   // Alarm 2: Door open request (Technoplat)
      dbx0_2 : Bool := FALSE;   // Alarm 3: Emergency push button (Technoplat)
      dbx0_3 : Bool := FALSE;   // Alarm 4: Thermic alarm (Technoplat)
      dbx0_4 : Bool := FALSE;   // Alarm 5: Fault inverters (Technoplat)
      dbx0_5 : Bool := FALSE;   // Alarm 6: Motor start missing (Technoplat)
      dbx0_6 : Bool := FALSE;   // Alarm 7: Stop cycle by operator (Technoplat)
      dbx0_7 : Bool := FALSE;   // Alarm 8: Film ended or broken (Technoplat)
      dbx1_0 : Bool := FALSE;   // Alarm 9: Machine table not in phase (Technoplat)
      dbx1_1 : Bool := FALSE;   // Alarm 10: The spool carriage encoder is not running (Technoplat)
      dbx1_2 : Bool := FALSE;   // Alarm 11: Table encoder not working well
      dbx1_3 : Bool := FALSE;   // Alarm 12: Overspeed for table rotation (Technoplat)
      dbx1_4 : Bool := FALSE;   // Alarm 13: Phase table sensor lost (Technoplat)
      dbx1_5 : Bool := FALSE;   // Alarm 14: table deceleration not correct (Technoplat)
      dbx1_6 : Bool := FALSE;   // Alarm 15: Pressure plate not up (Pressure plate)
      dbx1_7 : Bool := FALSE;   // Alarm 16: Timeout for pressure plate upward/downward (Pressure plate)
      dbx2_0 : Bool := FALSE;   // Alarm 17: Pallet lifter not down (Lifter)
      dbx2_1 : Bool := FALSE;   // Alarm 18: Timeout for pallet lifter upward/downward (Lifter)
      dbx2_2 : Bool := FALSE;   // Alarm 19: Wrong data program for the pallet on the machine (Technoplat)
      dbx2_3 : Bool := FALSE;   // Alarm 20: Sysdata error (Technoplat)
      dbx2_4 : Bool := FALSE;   // Alarm 21: Spool carriage not down (Technoplat)
      dbx2_5 : Bool := FALSE;   // Alarm 22: Pressure plate positioning lost during rotation
      dbx2_6 : Bool := FALSE;   // Alarm 23:
      dbx2_7 : Bool := FALSE;   // Alarm 24: Emergency on infeed safety barrier (Barrier)
      dbx3_0 : Bool := FALSE;   // Alarm 25: Emergency on outfeed safety barrier (Barrier)
      dbx3_1 : Bool := FALSE;   // Alarm 26: Safety barrier excluded in automatic mode (Barrier)
      dbx3_2 : Bool := FALSE;   // Alarm 27: Timeout for rope unit open/close (Rope unit)
      dbx3_3 : Bool := FALSE;   // Alarm 28: Timeout for full rope unit open/close (Rope unit)
      dbx3_4 : Bool := FALSE;   // Alarm 29:
      dbx3_5 : Bool := FALSE;   // Alarm 30: Profinet communication error
      dbx3_6 : Bool := FALSE;   // Alarm 31: Modbus communication error
      dbx3_7 : Bool := FALSE;   // Alarm 32:
      dbx4_0 : Bool := FALSE;   // Alarm 33: Pallet positioning released during table rotation (Conveyor
      dbx4_1 : Bool := FALSE;   // Alarm 34: Pallet in transit in infeed (Conveyor)
      dbx4_2 : Bool := FALSE;   // Alarm 35: Pallet in transit in outfeed (Conveyor)
      dbx4_3 : Bool := FALSE;   // Alarm 36: Wrong pallet positioning (Conveyor)
      dbx4_4 : Bool := FALSE;   // Alarm 37: Infeed ring rotation control engaged (Conveyor)
      dbx4_5 : Bool := FALSE;   // Alarm 38: Outfeed ring rotation control engaged (Conveyor)
      dbx4_6 : Bool := FALSE;   // Alarm 39: Technoplat table not in load phase
      dbx4_7 : Bool := FALSE;   // Alarm 40: Technoplat table not in unload phase
      dbx5_0 : Bool := FALSE;   // Alarm 41: Contrast carriage not back
      dbx5_1 : Bool := FALSE;   // Alarm 42: Timeout contrast carriage forward/backward
      dbx5_2 : Bool := FALSE;   // Alarm 43: Clamp not closed (Clamp)
      dbx5_3 : Bool := FALSE;   // Alarm 44: Welder contrast not down (Clamp)
      dbx5_4 : Bool := FALSE;   // Alarm 45: Welder unit not down (Clamp)
      dbx5_5 : Bool := FALSE;   // Alarm 46: Clamp not down (Clamp)
      dbx5_6 : Bool := FALSE;   // Alarm 47: Welder contrast not up (Clamp)
      dbx5_7 : Bool := FALSE;   // Alarm 48: Timeout for clamp open/close (Clamp)
      dbx6_0 : Bool := FALSE;   // Alarm 49: Timeout for clamp upward/downward (Clamp)
      dbx6_1 : Bool := FALSE;   // Alarm 50: Timeout for welder contrast upward/downward (Clamp)
      dbx6_2 : Bool := FALSE;   // Alarm 51: Timeout for welder unit upward/downward (Clamp)
      dbx6_3 : Bool := FALSE;   // Alarm 52: Check the welder circuit (Clamp)
      dbx6_4 : Bool := FALSE;   // Alarm 53: Welder and cut unit not backward (Clamp)
      dbx6_5 : Bool := FALSE;   // Alarm 54: Timeout for welder and cut unit forward/backward (Clamp)
      dbx6_6 : Bool := FALSE;   // Alarm 55: Timeout for clamp carriage forward/backward (Clamp)
      dbx6_7 : Bool := FALSE;   // Alarm 56: Clamp carriage not backward (Clamp)
      dbx7_0 : Bool := FALSE;   // Alarm 57: Top carriage not up (Top)
      dbx7_1 : Bool := FALSE;   // Alarm 58: Top carriage not backward (Top)
      dbx7_2 : Bool := FALSE;   // Alarm 59: Top cutter not backward (Top)
      dbx7_3 : Bool := FALSE;   // Alarm 60: Clamp to pull top film not open (Top)
      dbx7_4 : Bool := FALSE;   // Alarm 61: Clamp to block top film not closed (Top)
      dbx7_5 : Bool := FALSE;   // Alarm 62: Top carriage not in position (Top)
      dbx7_6 : Bool := FALSE;   // Alarm 63: Top carriage not inside top film cut area (Top)
      dbx7_7 : Bool := FALSE;   // Alarm 64: Safety for top carriage position (Top)
      dbx8_0 : Bool := FALSE;   // Alarm 65: Timeout for top cutter (Top)
      dbx8_1 : Bool := FALSE;   // Alarm 66: Timeout for clamp to pull top film (Top)
      dbx8_2 : Bool := FALSE;   // Alarm 67: Timeout for clamp to block top film (Top)
      dbx8_3 : Bool := FALSE;   // Alarm 68: Top film ended or broken (Top)
      dbx8_4 : Bool := FALSE;   // Alarm 69: Infeed safety for top carriage up/down (Top)
      dbx8_5 : Bool := FALSE;   // Alarm 70: Outfeed safety for top carriage up/down (Top)
      dbx8_6 : Bool := FALSE;   // Alarm 71: Clamp to blok top film not open (Top)
      dbx8_7 : Bool := FALSE;   // Alarm 72: Top rele' brake broken (Top)
      dbx9_0 : Bool := FALSE;   // Alarm 73: Top not in position (Top inside signal)
      dbx9_1 : Bool := FALSE;   // Alarm 74: LIFTER POS.2 EXTRASTROKE UP
      dbx9_2 : Bool := FALSE;   // Alarm 75: LIFTER POS.2 FOOT SAFETY
      dbx9_3 : Bool := FALSE;   // Alarm 76: LIFTER POS.2 TIMEOUT CONVEYOR
      dbx9_4 : Bool := FALSE;   // Alarm 77: LIFTER POS.2 TIMEOUT UPSTROKE
      dbx9_5 : Bool := FALSE;   // Alarm 78: LIFTER POS.2 TIMEOUT DOWNSTROKE
      dbx9_6 : Bool := FALSE;   // Alarm 79: LABEL FAULT
      dbx9_7 : Bool := FALSE;   // Alarm 80: Label not in home position with table rotation
      dbx10_0 : Bool := FALSE;   // Alarm 81: Fire door not open during pallet transit
      dbx10_1 : Bool := FALSE;   // Alarm 82:
      dbx10_2 : Bool := FALSE;   // Alarm 83:
      dbx10_3 : Bool := FALSE;   // Alarm 84:
      dbx10_4 : Bool := FALSE;   // Alarm 85:
      dbx10_5 : Bool := FALSE;   // Alarm 86:
      dbx10_6 : Bool := FALSE;   // Alarm 87:
      dbx10_7 : Bool := FALSE;   // Alarm 88:
      dbx11_0 : Bool := FALSE;   // Alarm 89:
      dbx11_1 : Bool := FALSE;   // Alarm 90:
      dbx11_2 : Bool := FALSE;   // Alarm 91:
      dbx11_3 : Bool := FALSE;   // Alarm 92:
      dbx11_4 : Bool := FALSE;   // Alarm 93:
      dbx11_5 : Bool := FALSE;   // Alarm 94:
      dbx11_6 : Bool := FALSE;   // Alarm 95:
      dbx11_7 : Bool := FALSE;   // Alarm 96:
      dbx12_0 : Bool := FALSE;   // Alarm 97:
      dbx12_1 : Bool := FALSE;   // Alarm 98:
      dbx12_2 : Bool := FALSE;   // Alarm 99:
      dbx12_3 : Bool := FALSE;   // Alarm 100:
      dbx12_4 : Bool := FALSE;   // Alarm 101:
      dbx12_5 : Bool := FALSE;   // Alarm 102:
      dbx12_6 : Bool := FALSE;   // Alarm 103:
      dbx12_7 : Bool := FALSE;   // Alarm 104:
      dbx13_0 : Bool := FALSE;   // Alarm 105:
      dbx13_1 : Bool := FALSE;   // Alarm 106:
      dbx13_2 : Bool := FALSE;   // Alarm 107:
      dbx13_3 : Bool := FALSE;   // Alarm 108:
      dbx13_4 : Bool := FALSE;   // Alarm 109:
      dbx13_5 : Bool := FALSE;   // Alarm 110:
      dbx13_6 : Bool := FALSE;   // Alarm 111:
      dbx13_7 : Bool := FALSE;   // Alarm 112:
      dbx14_0 : Bool := FALSE;   // Alarm 113:
      dbx14_1 : Bool := FALSE;   // Alarm 114:
      dbx14_2 : Bool := FALSE;   // Alarm 115:
      dbx14_3 : Bool := FALSE;   // Alarm 116:
      dbx14_4 : Bool := FALSE;   // Alarm 117:
      dbx14_5 : Bool := FALSE;   // Alarm 118:
      dbx14_6 : Bool := FALSE;   // Alarm 119:
      dbx14_7 : Bool := FALSE;   // Alarm 120:
      dbx15_0 : Bool := FALSE;   // Alarm 121:
      dbx15_1 : Bool := FALSE;   // Alarm 122:
      dbx15_2 : Bool := FALSE;   // Alarm 123:
      dbx15_3 : Bool := FALSE;   // Alarm 124:
      dbx15_4 : Bool := FALSE;   // Alarm 125:
      dbx15_5 : Bool := FALSE;   // Alarm 126:
      dbx15_6 : Bool := FALSE;   // Alarm 127:
      dbx15_7 : Bool := FALSE;   // Alarm 128:
      dbx16_0 : Bool := FALSE;   // Alarm 129:
      dbx16_1 : Bool := FALSE;   // Alarm 130:
      dbx16_2 : Bool := FALSE;   // Alarm 131:
      dbx16_3 : Bool := FALSE;   // Alarm 132:
      dbx16_4 : Bool := FALSE;   // Alarm 133:
      dbx16_5 : Bool := FALSE;   // Alarm 134:
      dbx16_6 : Bool := FALSE;   // Alarm 135:
      dbx16_7 : Bool := FALSE;   // Alarm 136:
      dbx17_0 : Bool := FALSE;   // Alarm 137:
      dbx17_1 : Bool := FALSE;   // Alarm 138:
      dbx17_2 : Bool := FALSE;   // Alarm 139:
      dbx17_3 : Bool := FALSE;   // Alarm 140:
      dbx17_4 : Bool := FALSE;   // Alarm 141:
      dbx17_5 : Bool := FALSE;   // Alarm 142:
      dbx17_6 : Bool := FALSE;   // Alarm 143:
      dbx17_7 : Bool := FALSE;   // Alarm 144:
      dbx18_0 : Bool := FALSE;   // Alarm 145:
      dbx18_1 : Bool := FALSE;   // Alarm 146:
      dbx18_2 : Bool := FALSE;   // Alarm 147:
      dbx18_3 : Bool := FALSE;   // Alarm 148:
      dbx18_4 : Bool := FALSE;   // Alarm 149:
      dbx18_5 : Bool := FALSE;   // Alarm 150:
      dbx18_6 : Bool := FALSE;   // Alarm 151:
      dbx18_7 : Bool := FALSE;   // Alarm 152:
      dbx19_0 : Bool := FALSE;   // Alarm 153:
      dbx19_1 : Bool := FALSE;   // Alarm 154:
      dbx19_2 : Bool := FALSE;   // Alarm 155:
      dbx19_3 : Bool := FALSE;   // Alarm 156:
      dbx19_4 : Bool := FALSE;   // Alarm 157:
      dbx19_5 : Bool := FALSE;   // Alarm 158:
      dbx19_6 : Bool := FALSE;   // Alarm 159:
      dbx19_7 : Bool := FALSE;   // Alarm 160:
      dbx20_0 : Bool := FALSE;   // Alarm 161:
      dbx20_1 : Bool := FALSE;   // Alarm 162:
      dbx20_2 : Bool := FALSE;   // Alarm 163:
      dbx20_3 : Bool := FALSE;   // Alarm 164:
      dbx20_4 : Bool := FALSE;   // Alarm 165:
      dbx20_5 : Bool := FALSE;   // Alarm 166:
      dbx20_6 : Bool := FALSE;   // Alarm 167:
      dbx20_7 : Bool := FALSE;   // Alarm 168:
      dbx21_0 : Bool := FALSE;   // Alarm 169:
      dbx21_1 : Bool := FALSE;   // Alarm 170:
      dbx21_2 : Bool := FALSE;   // Alarm 171:
      dbx21_3 : Bool := FALSE;   // Alarm 172:
      dbx21_4 : Bool := FALSE;   // Alarm 173:
      dbx21_5 : Bool := FALSE;   // Alarm 174:
      dbx21_6 : Bool := FALSE;   // Alarm 175:
      dbx21_7 : Bool := FALSE;   // Alarm 176:
      dbx22_0 : Bool := FALSE;   // Alarm 177:
      dbx22_1 : Bool := FALSE;   // Alarm 178:
      dbx22_2 : Bool := FALSE;   // Alarm 179:
      dbx22_3 : Bool := FALSE;   // Alarm 180:
      dbx22_4 : Bool := FALSE;   // Alarm 181:
      dbx22_5 : Bool := FALSE;   // Alarm 182:
      dbx22_6 : Bool := FALSE;   // Alarm 183:
      dbx22_7 : Bool := FALSE;   // Alarm 184:
      dbx23_0 : Bool := FALSE;   // Alarm 185:
      dbx23_1 : Bool := FALSE;   // Alarm 186:
      dbx23_2 : Bool := FALSE;   // Alarm 187:
      dbx23_3 : Bool := FALSE;   // Alarm 188:
      dbx23_4 : Bool := FALSE;   // Alarm 189:
      dbx23_5 : Bool := FALSE;   // Alarm 190:
      dbx23_6 : Bool := FALSE;   // Alarm 191:
      dbx23_7 : Bool := FALSE;   // Alarm 192:
      dbx24_0 : Bool := FALSE;   // Alarm 193:
      dbx24_1 : Bool := FALSE;   // Alarm 194:
      dbx24_2 : Bool := FALSE;   // Alarm 195:
      dbx24_3 : Bool := FALSE;   // Alarm 196:
      dbx24_4 : Bool := FALSE;   // Alarm 197:
      dbx24_5 : Bool := FALSE;   // Alarm 198:
      dbx24_6 : Bool := FALSE;   // Alarm 199:
      dbx24_7 : Bool := FALSE;   // Alarm 200:
      dbx25_0 : Bool := FALSE;   // Alarm 201:
      dbx25_1 : Bool := FALSE;   // Alarm 202:
      dbx25_2 : Bool := FALSE;   // Alarm 203:
      dbx25_3 : Bool := FALSE;   // Alarm 204:
      dbx25_4 : Bool := FALSE;   // Alarm 205:
      dbx25_5 : Bool := FALSE;   // Alarm 206:
      dbx25_6 : Bool := FALSE;   // Alarm 207:
      dbx25_7 : Bool := FALSE;   // Alarm 208:
      dbx26_0 : Bool := FALSE;   // Warning 1: %10 Prestretch film on spool carriage (Technoplat)
      dbx26_1 : Bool := FALSE;   // Warning 2:
      dbx26_2 : Bool := FALSE;   // Warning 3: Request to reset encoder on spool carriage (Technoplat)
      dbx26_3 : Bool := FALSE;   // Warning 4:
      dbx26_4 : Bool := FALSE;   // Warning 5: Request to reset encoder on table rotation (Technoplat)
      dbx26_5 : Bool := FALSE;   // Warning 6:
      dbx26_6 : Bool := FALSE;   // Warning 7:
      dbx26_7 : Bool := FALSE;   // Warning 8: Fire door closing request
      dbx27_0 : Bool := FALSE;   // Warning 9: Timeout for door opening
      dbx27_1 : Bool := FALSE;   // Warning 10:
      dbx27_2 : Bool := FALSE;   // Warning 11:
      dbx27_3 : Bool := FALSE;   // Warning 12:
      dbx27_4 : Bool := FALSE;   // Warning 13:
      dbx27_5 : Bool := FALSE;   // Warning 14:
      dbx27_6 : Bool := FALSE;   // Warning 15:
      dbx27_7 : Bool := FALSE;   // Warning 16:
      dbx28_0 : Bool := FALSE;   // Warning 17:
      dbx28_1 : Bool := FALSE;   // Warning 18:
      dbx28_2 : Bool := FALSE;   // Warning 19:
      dbx28_3 : Bool := FALSE;   // Warning 20:
      dbx28_4 : Bool := FALSE;   // Warning 21:
      dbx28_5 : Bool := FALSE;   // Warning 22:
      dbx28_6 : Bool := FALSE;   // Warning 23:
      dbx28_7 : Bool := FALSE;   // Warning 24:
      dbx29_0 : Bool := FALSE;   // Warning 25:
      dbx29_1 : Bool := FALSE;   // Warning 26:
      dbx29_2 : Bool := FALSE;   // Warning 27:
      dbx29_3 : Bool := FALSE;   // Warning 28:
      dbx29_4 : Bool := FALSE;   // Warning 29:
      dbx29_5 : Bool := FALSE;   // Warning 30:
      dbx29_6 : Bool := FALSE;   // Warning 31:
      dbx29_7 : Bool := FALSE;   // Warning 32:
   END_VAR
BEGIN
END_DATA_BLOCK

